// TwinCAT 3 PLC project STELLA1Runtime
// ProgramVersion: 3.1.4023.0
// libraries:
//   Tc2_DataExchange, * (Beckhoff Automation GmbH)
//   Tc2_Math, * (Beckhoff Automation GmbH)
//   Tc2_MC2, * (Beckhoff Automation GmbH)
//   Tc2_MC2_Drive, * (Beckhoff Automation GmbH)
//   Tc2_NC, * (Beckhoff Automation GmbH)
//   Tc2_Standard, * (Beckhoff Automation GmbH)
//   Tc2_System, * (Beckhoff Automation GmbH)
//   Tc2_Utilities, * (Beckhoff Automation GmbH)
//   Tc3_IotBase, * (Beckhoff Automation GmbH)
//   Tc3_Module, * (Beckhoff Automation GmbH)
//   VisuDialogs, * (System)
//   PS_DcUpsEC,2.0,Phoenix Contact GmbH & Co.KG
//   VisuSymbols,3.5.10.0,System
// project tree:
//   DUTs/ E_Blink.TcDUT (not stored), E_Horn.TcDUT (not stored), E_TCSCommand.TcDUT, E_TCSErrors.TcDUT, E_TelescopeMode.TcDUT (not stored)
//   / GlobalTextList.TcGTLO, PlcTask.TcTTO (not stored), Visualization Manager.TcVMO (not stored)
//   GVLs/ GVL_FilterWheel.TcGVL (not stored), GVL_Hydraulics.TcGVL, GVL_Main.TcGVL, GVL_pendant_control.TcGVL (not stored), GVL_Safety.TcGVL, GVL_Telescope.TcGVL (not stored)
//   POUs/ AzimuthElevationControl.TcPOU, CoverControl.TcPOU, DerotatorControl.TcPOU, ElevationControl.TcPOU, FilterWheelControl.TcPOU, FocusControl.TcPOU, HydraulicsControl.TcPOU, MAIN.TcPOU, NasmythControl.TcPOU (not stored), PendantControl.TcPOU (not stored), PowerMonitoring.TcPOU, SafetyHandling.TcPOU (not stored), TelescopeAuxiliary.TcPOU (not stored), TelescopeControl.TcPOU, Transformer.TcPOU
//   POUs/FunctionBlocks/ CO_ABERRATION.TcPOU, CO_NUTATE.TcPOU, CO_REFRACT.TcPOU (not stored), FB_ALTAZ2HADEC.TcPOU (not stored), FB_AstroClock.TcPOU, FB_Axis2.TcPOU, FB_BLINK.TcPOU, FB_ButtonEnable.TcPOU (not stored), FB_Cover.TcPOU (not stored), FB_CO_NUTATE.TcPOU (not stored), FB_EQ2HOR.TcPOU, FB_EQ2HOR2.TcPOU, FB_EventLog.TcPOU (not stored), FB_HADEC2ALTAZ.TcPOU (not stored), FB_HOR2EQ.TcPOU, FB_HOR2EQ2.TcPOU, FB_Horn.TcPOU, FB_InfluxMessage.TcPOU (not stored), FB_LightTimer.TcPOU, FB_MQTTCommunication.TcPOU, FB_NUTATE.TcPOU, FB_PRECESS.TcPOU (not stored), FB_PRECESS2.TcPOU (not stored), FB_PRECESS3.TcPOU, FB_RFTRIG.TcPOU (not stored), FB_SUNPOS.TcPOU, FB_TimeAverage.TcPOU, FB_Timer.TcPOU, FB_TONTP.TcPOU (not stored), TelescopeAxisClass.TcPOU (not stored)
//   POUs/Functions/ ATAN2.TcPOU, CO_REFRACT_FORWARD.TcPOU (not stored), CT2LST.TcPOU, DateTime2JD.TcPOU, F_Azimuthvelocity.TcPOU, F_DerotatorPosition2.TcPOU, F_Derotatorvelocity.TcPOU (not stored), F_Elevationvelocity.TcPOU, F_YREAL.TcPOU (not stored), NCError_TO_STRING.TcPOU, PointingModelAzimuth.TcPOU (not stored), PointingModelElevation.TcPOU (not stored), POLY.TcPOU, Refraction.TcPOU, TEN.TcPOU (not stored)
//   VISUs/ Visualization.TcVIS
// real-time tasks:
//   TASK PlcTask: cycle T#10ms, priority 20, ADS port 350
// motion (NC):
//   TASK NC-Task 1 SAF: cycle T#2ms, priority 4, ADS port 501
//   TASK NC-Task 1 SVB: cycle T#10ms, priority 8, ADS port 511
//   AXIS Fokus (id 1)
//     Dynamic: AccelerationMaximum=100, DecelerationMaximum=100, Acceleration=4.5, Deceleration=4.5, Jerk=13.5
//     Velo: RefSearch=0.2, RefSync=0.2, SlowManual=0.1, FastManual=0.5, Maximum=3
//     TargetPosControl: Range=0.1
//     OtherSettings: AllowMotionCmdToSlave=true, PulseDistancePos=1, PulseDistanceNeg=1
//     encoder EncType=4
//       EncPara: ScaleFactorNumerator=0.001, ScaleFactorDenominator=5, MaxCount=#x0000ffff
//         SoftEndMinControl: Enable=true
//         SoftEndMaxControl: Enable=true, Range=100
//         Inc: RefMode=2, RefSoftSyncMask=#x0000ffff
//     drive DrvType=23
//       Analog: VeloReferenz=10.2713178, VeloScale=10, TorqueSetpointScale=10, ScaleFactorActTorque=10
//       TimeComp: TaskDelayCycles=1
//     controller CtrType=1
//       CtrPara: PriorControlFactor=1
//         PosDiffControl: Range=1
//         PID: PosKp=12, CtrlOutputLimit=1
//         Observer: BandWidth=20
//   AXIS Derotator (id 2)
//     General: UnitName=°
//     Dynamic: AccelerationMaximum=20, DecelerationMaximum=20, Acceleration=3.70696, Deceleration=3.70696, Jerk=1.65107
//     Velo: RefSearch=1, RefSync=0.5, SlowManual=0.5, FastManual=5, Fast=11.7222517903646, Maximum=11.7223
//     PositionAreaControl: Range=10
//     TargetPosControl: Range=1, Time=0.1
//     OtherSettings: AllowMotionCmdToSlave=true
//     encoder EncType=8
//       EncPara: ScaleFactorNumerator=0.2, ScaleFactorDenominator=1048576, MaxCount=#xffffffff
//         SoftEndMinControl: Enable=true, Range=-70
//         SoftEndMaxControl: Enable=true, Range=380
//     drive DrvType=9
//       DrvPara: MaxCount=#xffffffff, DriveControlDWord=#x00030100
//         Analog: VeloReferenz=12.894476969401, TorqueSetpointScale=10, ScaleFactorActTorque=0.1
//         TimeComp: TaskDelayCycles=1
//     controller CtrType=1
//       CtrPara: PriorControlFactor=1
//         PosDiffControl: Range=1, Time=0.1
//         Observer: BandWidth=20
//   AXIS Azimuth (id 3)
//     General: UnitName=°
//     Dynamic: AccelerationMaximum=10, DecelerationMaximum=10, Acceleration=3, Deceleration=3, Jerk=1
//     Velo: RefSearch=2, RefSync=1, SlowManual=1, FastManual=5, Fast=798, Maximum=10
//     TargetPosControl: Range=1, Time=0.1
//     OtherSettings: AllowMotionCmdToSlave=true
//     encoder EncType=8
//       EncPara: ScaleFactorNumerator=360, ScaleFactorDenominator=1048576, MaxCount=#xffffffff
//         SoftEndMinControl: Enable=true, Range=-50
//         SoftEndMaxControl: Enable=true, Range=450
//         Inc: RefPosition=180, RefMode=2
//     drive DrvType=9
//       DrvPara: MaxCount=#xffffffff, DriveControlDWord=#x00030100
//         Analog: VeloReferenz=877.8, VeloScale=1.02400649589962, TorqueSetpointScale=10, ScaleFactorActTorque=0.1
//         TimeComp: TaskDelayCycles=1
//     controller CtrType=1
//       CtrPara: PriorControlFactor=1
//         PosDiffControl: Range=3, Time=0.1
//         Observer: BandWidth=20
//   AXIS Elevation (id 4)
//     General: UnitName=°
//     Dynamic: AccelerationMaximum=10, DecelerationMaximum=10, Acceleration=3, Deceleration=3, Jerk=2
//     Velo: RefSearch=0.5, RefSync=0.5, SlowManual=1, FastManual=3, Fast=1026, Maximum=10
//     TargetPosControl: Range=1, Time=0.1
//     OtherSettings: AllowMotionCmdToSlave=true
//     encoder EncType=8
//       EncPara: ScaleFactorNumerator=360, ScaleFactorDenominator=1048576, MaxCount=#xffffffff
//         SoftEndMinControl: Enable=true
//         SoftEndMaxControl: Enable=true, Range=91
//         Inc: RefPosition=73.9885, RefMode=2
//     drive DrvType=9
//       DrvPara: MaxCount=#xffffffff, DriveControlDWord=#x00030100
//         Analog: VeloReferenz=1128.6, VeloScale=1.02400649589962, TorqueSetpointScale=10, ScaleFactorActTorque=0.1
//         TimeComp: TaskDelayCycles=1
//     controller CtrType=1
//       CtrPara: PriorControlFactor=1
//         PosDiffControl: Range=1, Time=0.1
//         Observer: BandWidth=20
//   AXIS FilterWheel (id 5)
//     General: UnitName=°, UnitFlags=#x00000004
//     Dynamic: AccelerationMaximum=1500, DecelerationMaximum=1500, Acceleration=100, Deceleration=100, Jerk=100
//     Velo: RefSearch=5, RefSync=2.5, SlowManual=3, FastManual=30, Fast=207.666666666667, Maximum=207.667
//     TargetPosControl: Range=1
//     OtherSettings: AllowMotionCmdToSlave=true
//     encoder EncType=19
//       EncPara: ScaleFactorNumerator=10, ScaleFactorDenominator=1048576, MaxCount=#xffffffff
//         Inc: RefMode=1, HomingSensorSource=9
//     drive DrvType=16
//       DrvPara: MaxCount=#xffffffff, DriveControlDWord=#x00020000
//         Analog: VeloReferenz=228.433333333333, VeloScale=30, PosScale=10, TorqueSetpointScale=10, ScaleFactorActTorque=0.1
//         TimeComp: TaskDelayCycles=1
//     controller CtrType=1
//       CtrPara: PriorControlFactor=1
//         PosDiffControl: Enable=false, Range=0.2
//         PID: PosKp=5
//         Observer: BandWidth=20
// I/O:
//   DEVICE Gerät 1 (EtherCAT), AmsNetId 5.122.3.233.2.1
//     Klemme 30 (EK1200) [EK1200-5000 EtherCAT Netzteil (2A E-Bus)]
//       Safety Logic (EL6910) [EL6910, TwinSAFE PLC]
//       Safety IN (EL1904) [EL1904, 4 Ch. Safety Input 24V, TwinSAFE]
//         modules: Module 1 (FSOES)
//       Safety OUT (EL2904) [EL2904, 4 Ch. Safety Output 24V, 0.5A, TwinSAFE]
//         modules: Module 1 (FSOES), Module 2 (DO)
//       Power analysis (EL3443) [EL3443 3Ch. Power Measuring]
//       Power0 (EL9410) [EL9410 E-Bus Netzteilklemme (Diagnose)]
//       Main Panel IN (EL1008) [EL1008 8K. Dig. Eingang 24V, 3ms]
//       Hydraulics IN (EL1008) [EL1008 8K. Dig. Eingang 24V, 3ms]
//       Trafo Hydraulics IN (EL1008) [EL1008 8K. Dig. Eingang 24V, 3ms]
//       Main Panel Out (EL2008) [EL2008 8K. Dig. Ausgang 24V, 0.5A]
//       Trafo Hydraulics OUT (EL2008) [EL2008 8K. Dig. Ausgang 24V, 0.5A]
//       Temperature IN (EL3202) [EL3202 2K.Ana. Eingang PT100 (RTD)]
//       Power1 (EL9410) [EL9410 E-Bus Netzteilklemme (Diagnose)]
//       Pendant Control (EL1008) [EL1008 8K. Dig. Eingang 24V, 3ms]
//       Pendant Control2 (EL1008) [EL1008 8K. Dig. Eingang 24V, 3ms]
//       M2 M3 Limit switches (EL1008) [EL1008 8K. Dig. Eingang 24V, 3ms]
//       Cover Limit Switches (EL1008) [EL1008 8K. Dig. Eingang 24V, 3ms]
//       Telescope Hydraulics IN (EL1008) [EL1008 8K. Dig. Eingang 24V, 3ms]
//       Pendant Lights (EL2008) [EL2008 8K. Dig. Ausgang 24V, 0.5A]
//       Lock and Horn (EL2008) [EL2008 8K. Dig. Ausgang 24V, 0.5A]
//       Temperature M2 M1 (EL3064) [EL3064 4K.Ana. Eingang 0-10V]
//       Power2 (EL9410) [EL9410 E-Bus Netzteilklemme (Diagnose)]
//       FocusMotor (EL7342) [EL7342 2K. DC-Motor-Endstufe (50V, 3.5A)]
//       FocusEncoder (EL5101-0010) [EL5101-0010 1K. Inc. Encoder 5V (20 Mio. Inkremente/s)]
//       Cover Motors (EL2008) [EL2008 8K. Dig. Ausgang 24V, 0.5A]
//       Klemme 54 (EK1521) [EK1521 1-Port EtherCAT-Abzweig (FX-MultiMode)]
//         Klemme 55 (EK1501) [EK1501 EtherCAT-Koppler (2A E-Bus, FX-MultiMode, ID-Switch)]
//           FilterWheel (EL7211-0010) [EL7211-0010 1K. MDP742 Servo-Motor-Endstufe mit OCT (50V, 4,5A RMS)]
//           Klemme 57 (EL1008) [EL1008 8K. Dig. Eingang 24V, 3ms]
//           Klemme 58 (EL2008) [EL2008 8K. Dig. Ausgang 24V, 0.5A]
//           ShutterCOM (EL6001) [EL6001 Schnittstelle (RS232)]
//           Klemme 60 (EL3064) [EL3064 4K.Ana. Eingang 0-10V]
//           Klemme 69 (EL3202-0010) [EL3202-0010 2K. Ana. Eingang PT100 (RTD), hochgenau]
//           Klemme 65 (EL9011) [EL9011 Endklemme]
//       Klemme 61 (EK1110) [EK1110 EtherCAT-Verlängerung]
//     Derotator(AX5203-0000-0210) [AX5203-0000-0210 EtherCAT Drive (SoE, 2 Ch.)]
//     Azimuth (AX5125-0000-0214) [AX5125-0000-0214 EtherCAT Drive (SoE, 1 Ch.)]
//     Elevation (AX5125-0000-0214) [AX5125-0000-0214 EtherCAT Drive (SoE, 1 Ch.)]
//     Box 74 (Uninterruptible Power Supply) [QUINT4-UPS/24DC/24DC/40/EC]
// variable links:
//   Device 1 (EtherCAT) <-> Device 1 (EtherCAT)/Term 30 (EK1200)/Safety IN (EL1904)
//     Term 30 (EK1200)/Safety Logic (EL6910)/ConnectionOutputs/TwinSafeGroup1.Safety IN (EL1904) - Module 1 (FSOES)_10 RxPDO <-> Module 1 (FSOES)/TxPDO/FSOE
//   Device 1 (EtherCAT) <-> Device 1 (EtherCAT)/Term 30 (EK1200)/Safety Logic (EL6910)
//     Term 30 (EK1200)/Safety IN (EL1904)/Module 1 (FSOES)/RxPDO/FSOE <-> ConnectionInputs/TwinSafeGroup1.Safety IN (EL1904) - Module 1 (FSOES)_10 TxPDO
//     Term 30 (EK1200)/Safety OUT (EL2904)/Module 1 (FSOES)/TxPDO/FSOE <-> ConnectionOutputs/TwinSafeGroup1.Safety OUT (EL2904) - Module 1 (FSOES)_11 RxPDO
//   Device 1 (EtherCAT) <-> Device 1 (EtherCAT)/Term 30 (EK1200)/Safety OUT (EL2904)
//     Term 30 (EK1200)/Safety Logic (EL6910)/ConnectionInputs/TwinSafeGroup1.Safety OUT (EL2904) - Module 1 (FSOES)_11 TxPDO <-> Module 1 (FSOES)/RxPDO/FSOE
//   NC-Task 1 SAF/Axes/Azimuth <-> Device 1 (EtherCAT)/Azimuth (AX5125-0000-0214)
//     Drive/Inputs/In/nDataIn1 <-> AT/Following distance
//     Drive/Inputs/In/nDcOutputTime <-> InfoData/DcOutputShift
//     Drive/Inputs/In/nState1 <-> AT/Drive status word @bit 8
//     Drive/Inputs/In/nState2 <-> AT/Drive status word
//     Drive/Inputs/In/nState4 @bit 1 <-> WcState/InputToggle
//     Drive/Inputs/In/nState4 <-> WcState/WcState
//     Drive/Outputs/Out/nCtrl1 <-> MDT/Master control word @bit 8
//     Drive/Outputs/Out/nDataOut1 <-> MDT/Position command value
//     Enc/Inputs/In/nDataIn1 <-> AT/Position feedback 1 value
//     Enc/Inputs/In/nDataIn3 <-> AT/Probe value 1 positive edge
//     Enc/Inputs/In/nDcInputTime <-> InfoData/DcInputShift
//     Enc/Inputs/In/nState4 @bit 1 <-> WcState/InputToggle
//     Enc/Inputs/In/nState4 <-> WcState/WcState
//     Enc/Inputs/In/nState5 <-> AT/Probe 1 positive latched
//     Enc/Outputs/Out/nCtrl5 <-> MDT/Probe 1 enable
//   NC-Task 1 SAF/Axes/Derotator <-> Device 1 (EtherCAT)/Derotator(AX5203-0000-0210)
//     Drive/Inputs/In/nDataIn1 <-> AT 1/Following distance
//     Drive/Inputs/In/nDataIn3[0] <-> AT 1/Torque/force feedback value
//     Drive/Inputs/In/nDcOutputTime <-> InfoData/DcOutputShift
//     Drive/Inputs/In/nState1 <-> AT 1/Drive status word @bit 8
//     Drive/Inputs/In/nState2 <-> AT 1/Drive status word
//     Drive/Inputs/In/nState4 @bit 1 <-> WcState/InputToggle
//     Drive/Inputs/In/nState4 <-> WcState/WcState
//     Drive/Outputs/Out/nCtrl1 <-> MDT 1/Master control word @bit 8
//     Drive/Outputs/Out/nDataOut1 <-> MDT 1/Position command value
//     Enc/Inputs/In/nDataIn1 <-> AT 1/Position feedback 1 value
//     Enc/Inputs/In/nDcInputTime <-> InfoData/DcInputShift
//     Enc/Inputs/In/nState4 @bit 1 <-> WcState/InputToggle
//     Enc/Inputs/In/nState4 <-> WcState/WcState
//   NC-Task 1 SAF/Axes/Elevation <-> Device 1 (EtherCAT)/Elevation (AX5125-0000-0214)
//     Drive/Inputs/In/nDataIn1 <-> AT/Following distance
//     Drive/Inputs/In/nDcOutputTime <-> InfoData/DcOutputShift
//     Drive/Inputs/In/nState1 <-> AT/Drive status word @bit 8
//     Drive/Inputs/In/nState2 <-> AT/Drive status word
//     Drive/Inputs/In/nState4 @bit 1 <-> WcState/InputToggle
//     Drive/Inputs/In/nState4 <-> WcState/WcState
//     Drive/Outputs/Out/nCtrl1 <-> MDT/Master control word @bit 8
//     Drive/Outputs/Out/nDataOut1 <-> MDT/Position command value
//     Enc/Inputs/In/nDataIn1 <-> AT/Position feedback 1 value
//     Enc/Inputs/In/nDataIn3 <-> AT/Probe value 1 positive edge
//     Enc/Inputs/In/nDcInputTime <-> InfoData/DcInputShift
//     Enc/Inputs/In/nState4 @bit 1 <-> WcState/InputToggle
//     Enc/Inputs/In/nState4 <-> WcState/WcState
//     Enc/Inputs/In/nState5 <-> AT/Probe 1 positive latched
//     Enc/Outputs/Out/nCtrl5 <-> MDT/Probe 1 enable
//   NC-Task 1 SAF/Axes/FilterWheel <-> Device 1 (EtherCAT)/Term 30 (EK1200)/Term 54 (EK1521)/Term 55 (EK1501)/FilterWheel (EL7211-0010)
//     Drive/Inputs/In/nDcOutputTime <-> InfoData/DcOutputShift
//     Drive/Inputs/In/nState1 <-> DRV Statusword/Statusword
//     Drive/Inputs/In/nState2 <-> DRV Statusword/Statusword @bit 8
//     Drive/Inputs/In/nState4 @bit 1 <-> WcState/InputToggle
//     Drive/Inputs/In/nState4 <-> WcState/WcState
//     Drive/Inputs/In/nState8 <-> DRV Info data 1/Info data 1
//     Drive/Outputs/Out/nCtrl1 <-> DRV Controlword/Controlword
//     Drive/Outputs/Out/nCtrl2 <-> DRV Controlword/Controlword @bit 8
//     Drive/Outputs/Out/nDataOut2 <-> DRV Target velocity/Target velocity
//     Enc/Inputs/In/nDataIn1 <-> FB Position/Position
//     Enc/Inputs/In/nDcInputTime <-> InfoData/DcInputShift
//     Enc/Inputs/In/nState4 @bit 1 <-> WcState/InputToggle
//     Enc/Inputs/In/nState4 <-> WcState/WcState
//   NC-Task 1 SAF/Axes/Fokus <-> Device 1 (EtherCAT)/Term 30 (EK1200)/FocusEncoder (EL5101-0010)
//     Enc/Inputs/In/nDataIn1[0] <-> ENC Status compact/Counter value
//     Enc/Inputs/In/nDataIn2[0] <-> ENC Status compact/Latch value
//     Enc/Inputs/In/nState1 <-> ENC Status compact/Status/Latch C valid
//     Enc/Inputs/In/nState1 @bit 1 <-> ENC Status compact/Status/Latch extern valid
//     Enc/Inputs/In/nState1 @bit 6 <-> ENC Status compact/Status/Open circuit
//     Enc/Inputs/In/nState1 @bit 2 <-> ENC Status compact/Status/Set counter done
//     Enc/Inputs/In/nState1 @bit 5 <-> ENC Status compact/Status/Status of input status
//     Enc/Inputs/In/nState2 @bit 4 <-> ENC Status compact/Status/Status of extern latch
//     Enc/Inputs/In/nState2 <-> ENC Status compact/Status/Status of input A
//     Enc/Inputs/In/nState2 @bit 1 <-> ENC Status compact/Status/Status of input B
//     Enc/Inputs/In/nState2 @bit 2 <-> ENC Status compact/Status/Status of input C
//     Enc/Inputs/In/nState2 @bit 3 <-> ENC Status compact/Status/Status of input gate
//     Enc/Inputs/In/nState2 @bit 5 <-> ENC Status compact/Status/Sync error
//     Enc/Inputs/In/nState2 @bit 6 <-> ENC Status compact/Status/TxPDO State
//     Enc/Inputs/In/nState2 @bit 7 <-> ENC Status compact/Status/TxPDO Toggle
//     Enc/Inputs/In/nState4 @bit 1 <-> WcState/InputToggle
//     Enc/Inputs/In/nState4 <-> WcState/WcState
//     Enc/Outputs/Out/nCtrl1 <-> ENC Control compact/Control/Enable latch C
//     Enc/Outputs/Out/nCtrl1 @bit 3 <-> ENC Control compact/Control/Enable latch extern on negative edge
//     Enc/Outputs/Out/nCtrl1 @bit 1 <-> ENC Control compact/Control/Enable latch extern on positive edge
//     Enc/Outputs/Out/nCtrl1 @bit 2 <-> ENC Control compact/Control/Set counter
//     Enc/Outputs/Out/nDataOut1[0] <-> ENC Control compact/Set counter value
//   NC-Task 1 SAF/Axes/Fokus <-> Device 1 (EtherCAT)/Term 30 (EK1200)/FocusMotor (EL7342)
//     Drive/Inputs/In/nState1 @bit 3 <-> DCM Status Channel 1/Status/Error
//     Drive/Inputs/In/nState1 @bit 5 <-> DCM Status Channel 1/Status/Moving negative
//     Drive/Inputs/In/nState1 @bit 4 <-> DCM Status Channel 1/Status/Moving positive
//     Drive/Inputs/In/nState1 @bit 1 <-> DCM Status Channel 1/Status/Ready
//     Drive/Inputs/In/nState1 <-> DCM Status Channel 1/Status/Ready to enable
//     Drive/Inputs/In/nState1 @bit 6 <-> DCM Status Channel 1/Status/Torque reduced
//     Drive/Inputs/In/nState1 @bit 2 <-> DCM Status Channel 1/Status/Warning
//     Drive/Inputs/In/nState2 @bit 3 <-> DCM Status Channel 1/Status/Digital input 1
//     Drive/Inputs/In/nState2 @bit 4 <-> DCM Status Channel 1/Status/Digital input 2
//     Drive/Inputs/In/nState2 @bit 5 <-> DCM Status Channel 1/Status/Sync error
//     Drive/Inputs/In/nState2 @bit 7 <-> DCM Status Channel 1/Status/TxPDO Toggle
//     Drive/Inputs/In/nState4 @bit 1 <-> WcState/InputToggle
//     Drive/Inputs/In/nState4 <-> WcState/WcState
//     Drive/Outputs/Out/nCtrl1 <-> DCM Control Channel 1/Control/Enable
//     Drive/Outputs/Out/nCtrl1 @bit 2 <-> DCM Control Channel 1/Control/Reduce torque
//     Drive/Outputs/Out/nCtrl1 @bit 1 <-> DCM Control Channel 1/Control/Reset
//     Drive/Outputs/Out/nCtrl1 @bit 3 <-> DCM Control Channel 1/Control/Threshold active
//     Drive/Outputs/Out/nDataOut2[0] <-> DCM Velocity Channel 1/Velocity
//   STELLA1Runtime/STELLA1Runtime Instance <-> Device 1 (EtherCAT)/Azimuth (AX5125-0000-0214)
//     PlcTask Inputs/GVL_Telescope.Azimuth_diagnostic <-> AT/Diagnostic number
//     PlcTask Inputs/GVL_Telescope.Azimuth_inputs <-> AT/Digital inputs, state
//     PlcTask Inputs/GVL_Telescope.Azimuth_torque <-> AT/Torque/force feedback value
//   STELLA1Runtime/STELLA1Runtime Instance <-> Device 1 (EtherCAT)/Box 74 (Uninterruptible Power Supply)
//     PlcTask Inputs/MAIN.arrInputPD @bit {304..432 step 32} <-> TxPDO 1/BATTERY {1..5} ALARMS  (5 links)
//     PlcTask Inputs/MAIN.arrInputPD @bit 80 <-> TxPDO 1/STATUS ACTUAL INPUT CURRENT
//     PlcTask Inputs/MAIN.arrInputPD @bit 64 <-> TxPDO 1/STATUS ACTUAL INPUT VOLTAGE
//     PlcTask Inputs/MAIN.arrInputPD @bit 112 <-> TxPDO 1/STATUS ACTUAL OUTPUT CURRENT 1
//     PlcTask Inputs/MAIN.arrInputPD @bit 96 <-> TxPDO 1/STATUS ACTUAL OUTPUT VOLTAGE 1
//     PlcTask Inputs/MAIN.arrInputPD @bit 128 <-> TxPDO 1/STATUS BATTERY ACTUAL VOLTAGE
//     PlcTask Inputs/MAIN.arrInputPD @bit 144 <-> TxPDO 1/STATUS BATTERY CHARGE CURRENT
//     PlcTask Inputs/MAIN.arrInputPD @bit 160 <-> TxPDO 1/STATUS BATTERY TEMPERATURE
//     PlcTask Inputs/MAIN.arrInputPD @bit 176 <-> TxPDO 1/STATUS DEVICE TEMPERATURE
//     PlcTask Inputs/MAIN.arrInputPD <-> TxPDO 1/STATUS FUNCTIONS
//     PlcTask Inputs/MAIN.arrInputPD @bit 32 <-> TxPDO 1/STATUS INTERFACE
//     PlcTask Inputs/MAIN.arrInputPD @bit 192 <-> TxPDO 1/STATUS SOC REMAINING TIME
//     PlcTask Inputs/MAIN.arrInputPD @bit 224 <-> TxPDO 1/STATUS SOC REMAINING TIME PC SHUTDOWN
//     PlcTask Inputs/MAIN.arrInputPD @bit 240 <-> TxPDO 1/STATUS SOH REMAINING LIFETIME
//     PlcTask Inputs/MAIN.arrInputPD @bit 272 <-> TxPDO 1/UPS DIAGNOSIS ALARMS
//     PlcTask Inputs/MAIN.arrInputPD @bit 256 <-> TxPDO 1/UPS PROCESS ALARMS
//   STELLA1Runtime/STELLA1Runtime Instance <-> Device 1 (EtherCAT)/Derotator(AX5203-0000-0210)
//     PlcTask Inputs/GVL_Telescope.Derotator_diagnostic <-> AT 1/Diagnostic number
//     PlcTask Inputs/GVL_Telescope.Derotator_inputs <-> AT 1/Digital inputs, state
//     PlcTask Inputs/GVL_Telescope.Derotator_torque <-> AT 1/Torque/force feedback value
//   STELLA1Runtime/STELLA1Runtime Instance <-> Device 1 (EtherCAT)/Elevation (AX5125-0000-0214)
//     PlcTask Inputs/GVL_Telescope.Elevation_diagnostic <-> AT/Diagnostic number
//     PlcTask Inputs/GVL_Telescope.Elevation_inputs <-> AT/Digital inputs, state
//     PlcTask Inputs/GVL_Telescope.Elevation_torque <-> AT/Torque/force feedback value
//   STELLA1Runtime/STELLA1Runtime Instance <-> Device 1 (EtherCAT)/Term 30 (EK1200)/Cover Limit Switches (EL1008)
//     PlcTask Inputs/GVL_Telescope.cover1_closed <-> Channel 2/GVL_Telescope.cover1_closed
//     PlcTask Inputs/GVL_Telescope.cover2_closed <-> Channel 4/GVL_Telescope.cover2_closed
//     PlcTask Inputs/GVL_Telescope.cover3_closed <-> Channel 6/GVL_Telescope.cover3_closed
//     PlcTask Inputs/GVL_Telescope.cover1_open <-> Channel 1/GVL_Telescope.cover1_open
//     PlcTask Inputs/GVL_Telescope.cover2_open <-> Channel 3/GVL_Telescope.cover2_open
//     PlcTask Inputs/GVL_Telescope.cover3_open <-> Channel 5/GVL_Telescope.cover3_open
//   STELLA1Runtime/STELLA1Runtime Instance <-> Device 1 (EtherCAT)/Term 30 (EK1200)/Cover Motors (EL2008)
//     PlcTask Outputs/GVL_Telescope.close_cover1 <-> Channel 4/GVL_Telescope.close_cover1
//     PlcTask Outputs/GVL_Telescope.close_cover2 <-> Channel 6/GVL_Telescope.close_cover2
//     PlcTask Outputs/GVL_Telescope.close_cover3 <-> Channel 8/GVL_Telescope.close_cover3
//     PlcTask Outputs/GVL_Telescope.nasmyth_left <-> Channel 1/GVL_Telescope.nasmyth_left
//     PlcTask Outputs/GVL_Telescope.nasmyth_right <-> Channel 2/GVL_Telescope.nasmyth_right
//     PlcTask Outputs/GVL_Telescope.open_cover1 <-> Channel 3/GVL_Telescope.open_cover1
//     PlcTask Outputs/GVL_Telescope.open_cover2 <-> Channel 5/GVL_Telescope.open_cover2
//     PlcTask Outputs/GVL_Telescope.open_cover3 <-> Channel 7/GVL_Telescope.open_cover3
//   STELLA1Runtime/STELLA1Runtime Instance <-> Device 1 (EtherCAT)/Term 30 (EK1200)/Hydraulics IN (EL1008)
//     PlcTask Inputs/GVL_Hydraulics.oil_high <-> Channel 2/GVL_Hydraulics.oil_high
//     PlcTask Inputs/GVL_Hydraulics.oil_low <-> Channel 1/GVL_Hydraulics.oil_low
//     PlcTask Inputs/GVL_Hydraulics.oil_overtemperature <-> Channel 4/GVL_Hydraulics.oil_overtemperature
//     PlcTask Inputs/GVL_Hydraulics.oil_pressure_OK <-> Channel 3/GVL_Hydraulics.oil_pressure_OK
//     PlcTask Inputs/GVL_Hydraulics.oil_undertemperature <-> Channel 5/GVL_Hydraulics.oil_undertemperature
//     PlcTask Inputs/GVL_Hydraulics.oilfilter_dirty <-> Channel 6/GVL_Hydraulics.oilfilter_dirty
//   STELLA1Runtime/STELLA1Runtime Instance <-> Device 1 (EtherCAT)/Term 30 (EK1200)/Lock and Horn (EL2008)
//     PlcTask Outputs/GVL_Telescope.focus_unlock <-> Channel 1/GVL_Telescope.focus_lock
//     PlcTask Outputs/GVL_Telescope.horn <-> Channel 8/GVL_Telescope.horn
//     PlcTask Outputs/GVL_Telescope.nasmyth_lock <-> Channel 2/GVL_Telescope.nasmyth_lock
//   STELLA1Runtime/STELLA1Runtime Instance <-> Device 1 (EtherCAT)/Term 30 (EK1200)/M2 M3 Limit switches (EL1008)
//     PlcTask Inputs/GVL_Telescope.focus_limit_far <-> Channel 2/GVL_Telescope.focus_limit_far
//     PlcTask Inputs/GVL_Telescope.focus_limit_near <-> Channel 1/GVL_Telescope.focus_limit_near
//     PlcTask Inputs/GVL_Telescope.nasmyth_limit_left <-> Channel 3/GVL_Telescope.nasmyth_limit_left
//     PlcTask Inputs/GVL_Telescope.nasmyth_limit_right <-> Channel 4/GVL_Telescope.nasmyth_limit_right
//   STELLA1Runtime/STELLA1Runtime Instance <-> Device 1 (EtherCAT)/Term 30 (EK1200)/Main Panel IN (EL1008)
//     PlcTask Inputs/GVL_Main.key_switch_remote <-> Channel 1/GVL_Main.key_switch_remote
//     PlcTask Inputs/GVL_Main.reset_switch <-> Channel 4/GVL_Main.reset_switch
//     PlcTask Inputs/GVL_Main.start_switch <-> Channel 2/GVL_Main.start_switch
//     PlcTask Inputs/GVL_Main.stop_switch <-> Channel 3/GVL_Main.stop_switch
//   STELLA1Runtime/STELLA1Runtime Instance <-> Device 1 (EtherCAT)/Term 30 (EK1200)/Main Panel Out (EL2008)
//     PlcTask Outputs/GVL_Main.lamp_error <-> Channel 3/GVL_Main.lamp_error
//     PlcTask Outputs/GVL_Main.lamp_on_manual <-> Channel 2/GVL_Main.lamp_ready
//     PlcTask Outputs/GVL_Main.lamp_power <-> Channel 1/GVL_Main.lamp_power
//   STELLA1Runtime/STELLA1Runtime Instance <-> Device 1 (EtherCAT)/Term 30 (EK1200)/Pendant Control (EL1008)
//     PlcTask Inputs/GVL_pendant_control.BCD1 <-> Channel 1/GVL_pendant_control.BCD1
//     PlcTask Inputs/GVL_pendant_control.BCD2 <-> Channel 2/GVL_pendant_control.BCD2
//     PlcTask Inputs/GVL_pendant_control.BCD4 <-> Channel 3/GVL_pendant_control.BCD4
//     PlcTask Inputs/GVL_pendant_control.BCD8 <-> Channel 4/GVL_pendant_control.BCD8
//     PlcTask Inputs/GVL_pendant_control.direction_down <-> Channel 7/GVL_pendant_control.direction_down
//     PlcTask Inputs/GVL_pendant_control.direction_up <-> Channel 6/GVL_pendant_control.direction_up
//     PlcTask Inputs/GVL_pendant_control.key_switch <-> Channel 8/GVL_pendant_control.key_switch
//     PlcTask Inputs/GVL_pendant_control.reset_switch <-> Channel 5/GVL_pendant_control.reset_switch
//   STELLA1Runtime/STELLA1Runtime Instance <-> Device 1 (EtherCAT)/Term 30 (EK1200)/Pendant Control2 (EL1008)
//     PlcTask Inputs/GVL_pendant_control.direction_left <-> Channel 2/GVL_pendant_control.direction_left
//     PlcTask Inputs/GVL_pendant_control.direction_right <-> Channel 3/GVL_pendant_control.direction_right
//     PlcTask Inputs/GVL_pendant_control.start_switch <-> Channel 1/GVL_pendant_control.start_switch
//   STELLA1Runtime/STELLA1Runtime Instance <-> Device 1 (EtherCAT)/Term 30 (EK1200)/Pendant Lights (EL2008)
//     PlcTask Outputs/GVL_pendant_control.lamp_down <-> Channel 2/GVL_pendant_control.lamp_down
//     PlcTask Outputs/GVL_pendant_control.lamp_error <-> Channel 5/GVL_pendant_control.lamp_error
//     PlcTask Outputs/GVL_pendant_control.lamp_left <-> Channel 4/GVL_pendant_control.lamp_left
//     PlcTask Outputs/GVL_pendant_control.lamp_right <-> Channel 3/GVL_pendant_control.lamp_right
//     PlcTask Outputs/GVL_pendant_control.lamp_up <-> Channel 1/GVL_pendant_control.lamp_up
//   STELLA1Runtime/STELLA1Runtime Instance <-> Device 1 (EtherCAT)/Term 30 (EK1200)/Power analysis (EL3443)
//     PlcTask Inputs/GVL_Main.ActiveEnergy <-> Total Active/Active Energy
//     PlcTask Inputs/GVL_Main.ActivePower <-> Total Active/Active Power
//     PlcTask Inputs/GVL_Main.NeutralLineCurrent <-> Total Basic/Calculated Neutral Line Current
//   STELLA1Runtime/STELLA1Runtime Instance <-> Device 1 (EtherCAT)/Term 30 (EK1200)/Safety Logic (EL6910)
//     PlcTask Inputs/GVL_Safety.Error <-> StandardInputs/TwinSafeGroup1.SafetyError_4
//     PlcTask Inputs/GVL_Safety.State <-> Function Block Info Data/TwinSafeGroup1.Network1.FBEstop1 Info Data/State
//     PlcTask Inputs/GVL_Safety.Stop <-> StandardInputs/TwinSafeGroup1.SafetyStop_7
//     PlcTask Outputs/GVL_Safety.ErrAck <-> StandardOutputs/TwinSafeGroup1.ErrorAcknowledgement_1
//     PlcTask Outputs/GVL_Safety.Restart <-> StandardOutputs/TwinSafeGroup1.RestartSafety_2
//     PlcTask Outputs/GVL_Safety.Run <-> StandardOutputs/TwinSafeGroup1.RunSafety_3
//   STELLA1Runtime/STELLA1Runtime Instance <-> Device 1 (EtherCAT)/Term 30 (EK1200)/Telescope Hydraulics IN (EL1008)
//     PlcTask Inputs/GVL_Hydraulics.oil_reserve <-> Channel 2/GVL_Hydraulics.oil_reserve
//     PlcTask Inputs/GVL_Hydraulics.oilpan_maximum <-> Channel 1/GVL_Hydraulics.oilpan_maximum
//     PlcTask Inputs/GVL_Telescope.azimut_limit_switch <-> Channel 8/GVL_Telescope.azimut_limit_switch
//   STELLA1Runtime/STELLA1Runtime Instance <-> Device 1 (EtherCAT)/Term 30 (EK1200)/Temperature IN (EL3202)
//     PlcTask Inputs/GVL_Main.main_cabinet_temperature <-> RTD Inputs Channel 1/Value
//   STELLA1Runtime/STELLA1Runtime Instance <-> Device 1 (EtherCAT)/Term 30 (EK1200)/Temperature M2 M1 (EL3064)
//     PlcTask Inputs/GVL_Hydraulics.oil_level <-> AI Standard Channel 3/GVL_Hydraulics.oil_level
//     PlcTask Inputs/GVL_Telescope.temperature_mirror1 <-> AI Standard Channel 2/GVL_Telescope.temperature_mirror1
//     PlcTask Inputs/GVL_Telescope.temperature_mirror2 <-> AI Standard Channel 1/GVL_Telescope.temperature_mirror2
//   STELLA1Runtime/STELLA1Runtime Instance <-> Device 1 (EtherCAT)/Term 30 (EK1200)/Term 54 (EK1521)/Term 55 (EK1501)/FilterWheel (EL7211-0010)
//     PlcTask Inputs/GVL_FilterWheel.bCalibrationCam <-> DRV Info data 1/Info data 1
//   STELLA1Runtime/STELLA1Runtime Instance <-> Device 1 (EtherCAT)/Term 30 (EK1200)/Term 54 (EK1521)/Term 55 (EK1501)/Term 60 (EL3064)
//     PlcTask Inputs/TelescopeAuxiliary.raw_dewar_pressure <-> AI Standard Channel 1/Value
//   STELLA1Runtime/STELLA1Runtime Instance <-> Device 1 (EtherCAT)/Term 30 (EK1200)/Trafo Hydraulics IN (EL1008)
//     PlcTask Inputs/GVL_Hydraulics.pump_running <-> Channel 7/GVL_Hydraulics.pump_running
//     PlcTask Inputs/GVL_Hydraulics.suction_running <-> Channel 8/GVL_Hydraulics.suction_running
//     PlcTask Inputs/GVL_Main.brake_clearing <-> Channel 3/GVL_Main.brake_clearing
//     PlcTask Inputs/GVL_Main.trafo_bypassed <-> Channel 2/GVL_Main.trafo_bypassed
//   STELLA1Runtime/STELLA1Runtime Instance <-> Device 1 (EtherCAT)/Term 30 (EK1200)/Trafo Hydraulics OUT (EL2008)
//     PlcTask Outputs/GVL_Hydraulics.oil_pump_enable <-> Channel 1/GVL_Hydraulics.oil_pump_enable
//     PlcTask Outputs/GVL_Hydraulics.oil_suction_enable <-> Channel 2/GVL_Hydraulics.oil_suction_enable
//     PlcTask Outputs/GVL_Main.softstart_trafo <-> Channel 8/GVL_Main.softstart_trafo
//     PlcTask Outputs/GVL_Telescope.brake_azimuth_eve <-> Channel 3/GVL_Telescope.brake_azimuth_eve
//   STELLA1Runtime/STELLA1Runtime Instance <-> NC-Task 1 SAF/Axes/Azimuth
//     PlcTask Inputs/GVL_Telescope.AzimuthAxisRef.NcToPlc <-> Outputs/ToPlc
//     PlcTask Outputs/GVL_Telescope.AzimuthAxisRef.PlcToNc <-> Inputs/FromPlc
//   STELLA1Runtime/STELLA1Runtime Instance <-> NC-Task 1 SAF/Axes/Derotator
//     PlcTask Inputs/GVL_Telescope.DerotatorAxisRef.NcToPlc <-> Outputs/ToPlc
//     PlcTask Outputs/GVL_Telescope.DerotatorAxisRef.PlcToNc <-> Inputs/FromPlc
//   STELLA1Runtime/STELLA1Runtime Instance <-> NC-Task 1 SAF/Axes/Elevation
//     PlcTask Inputs/GVL_Telescope.ElevationAxisRef.NcToPlc <-> Outputs/ToPlc
//     PlcTask Outputs/GVL_Telescope.ElevationAxisRef.PlcToNc <-> Inputs/FromPlc
//   STELLA1Runtime/STELLA1Runtime Instance <-> NC-Task 1 SAF/Axes/FilterWheel
//     PlcTask Inputs/GVL_FilterWheel.FilterWheel_AxisRef.NcToPlc <-> Outputs/ToPlc
//     PlcTask Outputs/GVL_FilterWheel.FilterWheel_AxisRef.PlcToNc <-> Inputs/FromPlc
//   STELLA1Runtime/STELLA1Runtime Instance <-> NC-Task 1 SAF/Axes/Fokus
//     PlcTask Inputs/GVL_Telescope.FocusAxisRef.NcToPlc <-> Outputs/ToPlc
//     PlcTask Outputs/GVL_Telescope.FocusAxisRef.PlcToNc <-> Inputs/FromPlc

// ---- DUTs/E_TCSCommand.TcDUT
{attribute 'qualified_only'}
{attribute 'strict'}
TYPE E_TCSCommand :
(
	no_command := 0,
	gohome,
	park,
	track,
	goto,
	stop,
	slew,
	poweron
);
END_TYPE

// ---- DUTs/E_TCSErrors.TcDUT
{attribute 'qualified_only'}
{attribute 'strict'}
TYPE E_TCSErrors :
(
	no_error := 0,
	info :=1,
	warning := 2,
    error := 4,
	panic := 8
);
END_TYPE

// ---- GVLs/GVL_Hydraulics.TcGVL
{attribute 'qualified_only'}
VAR_GLOBAL
	// 2.1
	oil_low				AT%I*: BOOL;
	// ?
	oil_high			AT%I*: BOOL;
	// 2.3
	oil_pressure_OK		AT%I*: BOOL;
	// 2.4
	oil_overtemperature		AT%I*: BOOL;
	// 2.5
	oil_undertemperature	AT%I*: BOOL;
	// 2.6
	oilfilter_dirty		AT%I*: BOOL;
	// 2.7
	pump_running		AT%I*: BOOL;
	// 2.8
	suction_running		AT%I*: BOOL;
	//BT2
	oil_level			AT%I*: INT;
	
	//DIN39 4.6
	oilpan_maximum		AT%I*: BOOL;
	//DIN40 4.7
	oil_reserve			AT%I*: BOOL;
	
		
	//DOUT4 0.3
	oil_pump_enable		AT%Q*: BOOL;
	//DOUT5 0.4
	oil_suction_enable		AT%Q*: BOOL;	
END_VAR

// ---- GVLs/GVL_Main.TcGVL
{attribute 'qualified_only'}
//TODO update to current RoboTel IOs
VAR_GLOBAL
	//DIN1 0.0
	//phase_available		AT%I*: BOOL;
	// not implemented on stella
	trafo_bypassed		AT%I*: BOOL;
	//not implemented on RoboTel
	//key_switch			AT%I*: BOOL;
	//DIN3 0.2
	key_switch_remote	AT%I*: BOOL;
	//DIN4 0.3
	start_switch		AT%I*: BOOL;
	//DIN5 0.4
	stop_switch			AT%I*: BOOL;
	//DIN8 0.7
	reset_switch		AT%I*: BOOL;
	
	//BT1
	main_cabinet_temperature	AT%I*: INT;
	//DIN15 1.6
	brake_clearing		AT%I*: BOOL;
	
	//DOUT1 0.0
	lamp_power			AT%Q*: BOOL;
	//DOUT2 0.1
	lamp_on_manual			AT%Q*: BOOL;
	//DOUT3 0.2
	lamp_error			AT%Q*: BOOL;
	
	//DOUT7 0.6
	softstart_trafo		AT%Q*:BOOL;

	isRoboTel:		BOOL;
	(*
	NeutralCurrentGuardWarning		AT%I*:	BOOL;
	NeutralCurrentGuarError			AT%I*:	BOOL;
	ActivePowerGuardWarning			AT%I*:	BOOL;
	ActivePowerGuardError			AT%I*:	BOOL;
	ApparentPowerGuardWarning		AT%I*:	BOOL;
	ApparentPowerGuardError			AT%I*:	BOOL;
	*)
END_VAR

// ---- GVLs/GVL_Safety.TcGVL
{attribute 'qualified_only'}
VAR_GLOBAL
	// Safety Error Condition
	Error		AT%I*:	BOOL;
	// Run/Stop Safety
	Run			AT%Q*:	BOOL;
	// Restart Safety
	Restart		AT%Q*:	BOOL;
	// Error Acknowledgement 
	ErrAck		AT%Q*:	BOOL;
	// Stop signal coming from Safety
	Stop		AT%I*:	BOOL;
	// state variable
	State		AT%I*:	USINT;
END_VAR

// ---- POUs/AzimuthElevationControl.TcPOU
PROGRAM AzimuthElevationControl
VAR_INPUT
	// enable the axis and its position control loop
	Enable:		BOOL;
	// reset the axis
	Reset: 		BOOL;
	// decrease azimuth
	left:		BOOL;
	// increase azimuth
	right: 		BOOL;
	// Move azimuth to given position
	MoveAxis:	BOOL;
	// Home the axis
	HomeAxis:	BOOL;
	// enable tracking
	Tracking:	BOOL;
	// position to move the axis to
	position: 	LREAL;
	// set the Velocity of the axis
	velocity:	LREAL;
	// stop the Axis
	StopAxis:	BOOL;
	// diagnostic reset
	bSoEReset:	BOOL;
END_VAR
VAR_OUTPUT
	// error state of the axis
	error: 			BOOL;
	// error ID of the axis
	ErrorID:		UDINT;
	// actual_position of the axis
	act_position:	LREAL;
	// is the axis calibrated
	calibrated:		BOOL;
	// drive is ready
	ready:			BOOL;
	// time to reach target position
	slewtime:		LREAL;
END_VAR
VAR
	AzimuthAxis:		FB_Axis2;
	AzimuthCalibration: MC_SetPosition;
	//fbSoEReset:			FB_SoEReset;
	AzimuthAxisEvent: 	FB_EventLog;
	AzimuthDiagnosticEvent: 	FB_EventLog;
	// delay until commutator angle is measured
	readydelay:			TON;
	HomeDelay:			FB_TONTP;
	TorqueError:		TON := (PT := T#3S);
	azimuth_torque: 	REAL;
	TorqueWarning:		FB_EventLog;
	CalibrationEvent:	FB_Eventlog;
	ReadParameter:		MC_ReadParameter;
	getlastposition:	BOOL := TRUE;
	azimuth_rest_timer:	TON;
	azimuth_at_rest:	BOOL;
	fbSoEReset: 		FB_SoEReset;
	DiagnosticError:	BOOL;
END_VAR
VAR CONSTANT
	// reference position for homing
	// homing_position:		LREAL := 439.0; // was 442 - -21.21 = 463.21; 463 + 24 = 439
	// current position of the calibration cam encoder zero index. Apply an offset here if necessary
	calibration_position:	LREAL :=  208.5009; //208.4983 - -0.0026;//208.6273; //208.6073; // 208.7122869;//207.0092; // 208.2342; 
END_VAR
VAR PERSISTENT
	last_position:	LREAL := -51.0;
END_VAR

(* Azimuth Axis control section
Power must be on and brake must be open for the axis to operate
*)

// generate the ready signal after enabling the drive
readydelay(IN :=  AzimuthAxis.Enable, PT := T#3000MS, Q=> ready);

// limit the input position angle
position := LIMIT(-50.0, position, 450.0);

// conduct the calibrated signal
calibrated := AzimuthAxis.Calibrated;

IF Calibrated OR Error THEN
	HomeAxis := FALSE;
	getlastposition := FALSE;
END_IF
	
IF HomeAxis THEN
	position := calibration_position;
END_IF

IF HomeDelay.Q THEN
	position := calibration_position;
	MoveAxis := TRUE;
END_IF

// perform a recalibration on the last known position
AzimuthCalibration(
	Axis := GVL_Telescope.AzimuthAxisRef,
	Execute := getlastposition AND last_position>=-50.0 AND NOT Calibrated,
	Position := last_position);

IF AzimuthCalibration.Done THEN
	getlastposition := FALSE;
END_IF

IF Calibrated THEN
	last_position := act_position;
END_IF

// enable the azimuth if not moved by the power chain. Sorry for the hack
azimuth_rest_timer(IN := HydraulicsControl.brake_open AND 
				(ABS(GVL_Telescope.AzimuthAxisRef.NcToPlc.ActVelo) < 0.01), PT := T#2S);
// if azimuth at rest or calibrated, allow enabling the azimuth
IF azimuth_rest_timer.Q or calibrated THEN
	azimuth_at_rest := TRUE;
ELSIF HydraulicsControl.brake_closed THEN
	azimuth_at_rest := FALSE;
END_IF
	
// deactivate limit switches on homing
MC_SetAcceptBlockedDriveSignal(
	Axis := GVL_Telescope.AzimuthAxisRef, 
	Enable := HomeAxis);

AzimuthAxis(	
	Enable := 			enable AND azimuth_at_rest AND NOT GVL_Telescope.azimut_limit_switch,
	Reset := 			reset,
	MoveAxis :=			MoveAxis,
	HomeAxis := 		HomeAxis,
	StopAxis :=			StopAxis,
	Tracking :=			Tracking,
	Position := 		position, 
	Velocity :=			velocity,
	Enable_Positive := 	GVL_Telescope.Azimuth_inputs.1 OR HomeAxis,
	Enable_Negative := 	GVL_Telescope.Azimuth_inputs.0,
	Jog_Forward :=		right,
	Jog_Backwards := 	left,
	bCalibrationCam :=	NOT GVL_Telescope.Azimuth_inputs.1,
	ActualPosition => 	act_position,
	Error => 			error,
	ErrorID => 			ErrorID,
	AxisRef :=			GVL_Telescope.AzimuthAxisRef);

IF bSoEReset THEN
	last_position := -51.0;
	fbSoEReset(
		Axis := GVL_Telescope.AzimuthAxisRef,
		Execute := TRUE,
		Timeout := DEFAULT_ADS_TIMEOUT);
 	IF fbSoEReset.Busy THEN
		fbSoEReset(Axis := GVL_Telescope.AzimuthAxisRef, Execute := FALSE);
	ELSE
		bSoEReset := FALSE;
		Reset := TRUE;
	END_IF
END_IF 

IF AzimuthAxis.MoveDone THEN
	MoveAxis := FALSE;
END_IF

IF AzimuthAxis.HomeDone THEN
	HomeAxis := FALSE;
END_IF
	
IF AzimuthAxis.ResetDone THEN
	reset := FALSE;
END_IF

IF AzimuthAxis.StopDone THEN
	StopAxis := FALSE;
END_IF
DiagnosticError := FALSE;
IF GVL_Telescope.Azimuth_diagnostic < 16#D012 AND GVL_Telescope.Azimuth_diagnostic > 16#D014 THEN
	DiagnosticError :=TRUE;
	ErrorID := GVL_Telescope.Azimuth_diagnostic;
END_IF

ReadParameter(	Axis := GVL_Telescope.AzimuthAxisRef, Enable := AzimuthAxis.InMotion, 
				ParameterNumber := MC_AxisParameter.AxisRemainingTimeToGo, 
				ReadMode := E_ReadMode.READMODE_CYCLIC);
IF ReadParameter.Valid THEN
	slewtime := ReadParameter.Value;
END_IF

azimuth_torque := GVL_Telescope.Azimuth_torque / 10.0;
TorqueError(IN := ABS(azimuth_torque) > 50.0);


AzimuthAxisEvent(	
	Trigger := 		Error, 
	Level := 		ADSLOG_MSGTYPE_ERROR,
	FormatString :=	'Azimuth Axis Error: %s',
	OnMessage := 	NCError_TO_STRING(ErrorID));
	
AzimuthDiagnosticEvent(	
	Trigger := 		DiagnosticError,
	Level := 		ADSLOG_MSGTYPE_ERROR,
	FormatString :=	'Azimuth Axis Diagnostic Error: %s',
	OnMessage := 	NCError_TO_STRING(GVL_Telescope.Azimuth_diagnostic));
	
TorqueWarning(	
	Trigger := 		TorqueError.Q, 
	Level := 		ADSLOG_MSGTYPE_WARN,
	FormatString :=	'%s',
	OnMessage := 	'Azimuth torque is high.');
	
CalibrationEvent(
	Trigger := 		Calibrated, 
	Level := 		ADSLOG_MSGTYPE_HINT,
	FormatString :=	'%s',
	OnMessage := 	'Azimuth axis is calibrated.');

END_PROGRAM

// ---- POUs/FunctionBlocks/FB_Axis2.TcPOU
FUNCTION_BLOCK FB_Axis2
VAR_INPUT
	// enable the axis
	Enable:		BOOL;
	// reset the axis after error
	Reset: 		BOOL;
	// Move the Axis to a given position
	MoveAxis: 	BOOL;
	// HomeAxis;
	HomeAxis:	BOOL;
	// Stop the axis
	StopAxis:	BOOL;
	// position to move to
	Position: 	LREAL;
	// maximum velocity
	Velocity:	LREAL := 10.0;
	// Enable movement in positive direction (considering limit switch)
	Enable_Positive:	BOOL := TRUE;
	// Enable movement in negative direction (considering limit switch)
	Enable_Negative:	BOOL := TRUE;
	// jog forward
	Jog_Forward:		BOOL := FALSE;
	// jog backward
	Jog_Backwards:		BOOL := FALSE;
	// calibration input for homing
	bCalibrationCam:	BOOL;
	isModuloAxis:		BOOL := FALSE;
	// enable external setpoint generator
	Tracking:			BOOL;
	HomingMode:			MC_HomingMode := MC_HomingMode.MC_DefaultHoming;
END_VAR
VAR_OUTPUT
	// Reset has been executed
	ResetDone:	BOOL; 
	// the axis is in target position
	MoveDone:	BOOL;
	// the axis hass jogged
	JogDone:	BOOL;
	// the axis has stopped
	StopDone: 	BOOL;
	// the axis was calibrated and has come to a standstill
	HomeDone:	BOOL;
	// the axis is ready
	Ready:		BOOL;
	// the command has been aborted
	CommandAborted: BOOL;
	// axis busy
	Busy: 		BOOL;
	// axis is moving
	Active: 	BOOL;
	// axis is stopping
	Stopping:	BOOL;
	// axis is standing still (no commands issued) this should be the default
	StandStill:	BOOL;
	// axis is in motion
	InMotion:	BOOL;
	// axis is homing
	Homing:		BOOL;
	// axis is Accelerating or Decelerating
	InRamp:		BOOL;
	// axis is tracking on position
	isTracking:	BOOL;
	//	error condition
	Error: 		BOOL;
	// number of error
	ErrorID: 	UDINT;
	// actual position of the axis
	ActualPosition: LREAL;
	// axis is calibrated;
	Calibrated:	BOOL := FALSE;
	
END_VAR
VAR
	Axis_Power:		MC_Power;
	Axis_Reset:		MC_Reset;
	Axis_Move:		MC_MoveAbsolute;
	Axis_Modulo:	MC_MoveModulo;
	//Axis_Position:	MC_ReadActualPosition;
	Axis_Stop:		MC_Stop;
	Axis_Status:	MC_ReadStatus;
	Axis_Home:		MC_Home;
	Axis_Jog: 		MC_Jog;
	Axis_SetpointEnable:	MC_ExtSetPointGenEnable;
	Axis_SetpointDisable:	MC_ExtSetPointGenDisable;
	StopAllowed:	BOOL;
	// Direction for Axis_SetpointFeed
	Direction:			DINT;
	// difference between set position and measured position
	PositionDifference:	LREAL;
	TrackPosition:		LREAL;
	TrackVelocity:		LREAL;
	TrackAcceleration:	LREAL;
END_VAR

VAR_IN_OUT
	// axis reference
	AxisRef:	AXIS_REF;
END_VAR

// query the status of the axis at the beginning of the cycle
Axis_Status(Enable := TRUE,
			Axis := AxisRef);

// Enable the axis (power signal or manual enable)
Axis_Power(
	Axis := AxisRef,
	Enable := Enable,
	Enable_Positive := Enable_Positive,
	Enable_Negative := Enable_Negative,
	Override := 100.0,
	Status => Ready);

Axis_Reset(
	Axis := 	AxisRef,
	Execute := 	Reset,
	Done => 	ResetDone);

(* Tracking section ********************************************** *)

IF Tracking THEN
	PositionDifference := LIMIT(-0.02, Position - ActualPosition, 0.02);
	TrackPosition := ActualPosition + PositionDifference;
	TrackVelocity := 0.0; // LIMIT(-1.0, 2.0 * Velocity, 1.0);
	TrackAcceleration := 0.0;
ELSE
	TrackPosition := ActualPosition;
	TrackVelocity := 0.0;
	TrackAcceleration := 0.0;
END_IF


IF NOT Tracking OR ABS(PositionDifference) < 1E-5 THEN // TrackVelocity = 0 AND TrackAcceleration = 0 THEN
	Direction := 0;
ELSIF PositionDifference < 0.0 THEN
	Direction := -1;
ELSE
	Direction := 1;
END_IF

isTracking := Tracking AND ABS(Position - ActualPosition) < 5.0E-3;
IF Tracking AND Ready AND Calibrated AND NOT StopAxis THEN
	Axis_SetpointEnable.Execute := TRUE;
ELSIF NOT Axis_SetpointEnable.Busy AND Axis_SetpointEnable.Done THEN
	Axis_SetpointEnable.Execute := FALSE;
END_IF

Axis_SetpointEnable(Axis := AxisRef,
	Position :=		TrackPosition,	// final destination
	PositionType := POSITIONTYPE_ABSOLUTE);
	
MC_ExtSetPointGenFeed(
	Position :=		TrackPosition,
	Velocity :=		TrackVelocity,
	Acceleration :=	TrackAcceleration,
	Direction :=	Direction, 
	Axis :=			AxisRef);

Axis_SetpointDisable(Axis := AxisRef,
	Execute := NOT Tracking);
	
(* end of tracking section  ********************************************** *)
	
IF isModuloAxis THEN
	Axis_Modulo( 
		Axis := 		AxisRef,
		Execute := 		MoveAxis AND Ready AND Calibrated,
		Position := 	Position,
		Velocity :=		Velocity,
		Direction := 	MC_Shortest_Way,
		Done => 		MoveDone);
ELSE
	Axis_Move( 
		Axis := 		AxisRef,
		Execute := 		MoveAxis AND Ready AND Calibrated,
		Position := 	Position,
		Velocity := 	Velocity,
		Done => 		MoveDone);
END_IF

Axis_Jog(
	JogForward := 	Jog_Forward AND Ready AND Enable_Positive,
	JogBackwards := Jog_Backwards AND Ready AND Enable_Negative,
	Mode := 		MC_JOGMODE_STANDARD_FAST,
	Done => 		JogDone, 
	Axis := 		AxisRef);

Axis_Home(
	Axis := 			AxisRef,
	Execute := 			HomeAxis AND Ready,
	Position := 		position, //DEFAULT_HOME_POSITION,
	HomingMode :=		HomingMode,
	bCalibrationCam := 	bCalibrationCam,
	Done => 			HomeDone);	
(*	
IF (MoveDone OR HomeDone OR JogDone) AND NOT Axis_Status.StandStill THEN
	StopAxis := TRUE;
END_IF
*)
IF MoveDone AND (NOT Axis_Modulo.Busy OR NOT Axis_Move.Busy) THEN
	MoveAxis := FALSE;
END_IF

IF JogDone THEN
	Jog_Forward := FALSE;
	Jog_Backwards := FALSE;
END_IF

IF HomeDone THEN
	Calibrated := TRUE;
	HomeAxis := FALSE;
END_IF

IF StopDone THEN
	StopAxis := FALSE;
END_IF

StopAllowed :=	Axis_Status.StandStill OR  
				Axis_Status.ContinuousMotion OR
				Axis_Status.DiscreteMotion OR
				Axis_Status.SynchronizedMotion OR
				Axis_Status.Homing;

Axis_Stop( 
	Axis := 	AxisRef,
	Execute := 	StopAxis AND StopAllowed,
	Done => 	StopDone);
(*
Axis_Position(
	Axis := 	AxisRef,
	Enable := 	Calibrated,
	Position => AbsolutePosition);
*)
IF isModuloAxis THEN
	ActualPosition := AxisRef.NcToPlc.ModuloActPos; // required e.g. for Filterwheel
ELSE
	ActualPosition := AxisRef.NcToPlc.ActPos;
END_IF

IF Axis_Power.Error THEN
	ErrorID := Axis_Power.ErrorID;
END_IF

IF Axis_SetpointEnable.Error THEN
	ErrorID := Axis_SetpointEnable.ErrorID;
END_IF

IF Axis_Reset.Error THEN
	ErrorID := Axis_Reset.ErrorID;
END_IF

IF Axis_Modulo.Error THEN
	ErrorID := Axis_Modulo.ErrorID;
END_IF

IF Axis_Move.Error THEN
	ErrorID := Axis_Move.ErrorID;
END_IF

IF Axis_Home.Error THEN
	ErrorID := Axis_Home.ErrorID;
END_IF

IF Axis_Jog.Error THEN
	ErrorID := Axis_Jog.ErrorID;
END_IF

IF Axis_Stop.Error THEN
	ErrorID := Axis_Stop.ErrorID;
END_IF

Busy := 	Axis_SetpointEnable.Busy OR
			Axis_Reset.Busy OR 
			Axis_Modulo.Busy OR
			Axis_Move.Busy OR 
			Axis_Home.Busy OR
			Axis_Jog.Busy;

Error := 	Axis_Power.Error OR 
			Axis_SetpointEnable.Error OR
			Axis_Reset.Error OR 
			Axis_Modulo.Error OR
			Axis_Move.Error OR 
			Axis_Home.Error OR
			Axis_Jog.Error OR 
			Axis_Stop.Error;

Active := 	// Axis_Power.Active OR //alsways true if enabled 
			Axis_Modulo.Active OR
			Axis_Move.Active OR 
			Axis_Home.Active OR
			Axis_Jog.Active OR 
			Axis_Stop.Active;

CommandAborted :=	Axis_Modulo.CommandAborted OR
					Axis_Move.CommandAborted OR 
					Axis_Home.CommandAborted OR
					Axis_Jog.CommandAborted OR 
					Axis_Stop.CommandAborted;	
	
IF NOT Error THEN
	ErrorID := 0;
END_IF
			
InMotion := Axis_Status.ConstantVelocity OR
			Axis_Status.DiscreteMotion OR
			Axis_Status.ContinuousMotion OR
			Axis_Status.SynchronizedMotion; 
InRamp :=	Axis_Status.Accelerating OR
			Axis_Status.Decelerating;
Stopping := Axis_Status.Stopping;
StandStill := Axis_Status.StandStill;
Homing :=	Axis_Status.Homing;
// InPosition := AxisRef.NcToPlc.TargetPos;

END_FUNCTION_BLOCK

// ---- POUs/HydraulicsControl.TcPOU
PROGRAM HydraulicsControl
VAR_INPUT
	// start the hydraulics
	enable:		BOOL := FALSE;
	// reset any hydraulics error
	reset: 		BOOL;
	// manual override to start the suction pump
	suction_manual:	BOOL;
	//manual override to stop the pump
	pump_manual_stop: BOOL;
END_VAR
VAR_OUTPUT
	// status of the brake: is the brake open?
	brake_open:			BOOL;
	// is the brake closed?
	brake_closed:		BOOL;
	// pump is running, but the pressure remains low
	pressure_failure:	BOOL;
	// suction was started, but it is not running
	suction_failure:	BOOL;
	// main pump is running but suction has a timeout
	hydraulics_failure:	BOOL;
	main_pump_failure: BOOL;
	// oil is low
	oil_low:			BOOL;
	// oil is high (unused?)
	oil_high:			BOOL;
	// oil pressure is 25 bars
	oil_pressure_OK:	BOOL;
	// oil is on reserve
	oil_warning:		BOOL;
	// oil filter is dirty
	oil_filter_dirty:	BOOL;
	// oil is below 10°C
	oil_cold:			BOOL;
	// oil is above 50°C
	oil_hot:			BOOL;
	// main pump is running
	pump_running:		BOOL;
	// suction pump is running
	suction_running :	BOOL := FALSE;
	// error condition
	error: 				BOOL;
END_VAR
VAR
	// command to open the brake
	iopen_brake:	BOOL := FALSE;
	// command to open the brake
	iclose_brake: BOOL;
	// monitors the pressure of the pump is running
	pressure_watchdog:	TON;
	// monitors the activation of the suction pump
	suction_watchdog: TON;
	// monitors the activation of the main pump
	main_pump_watchdog:	TON;
	// watch the hydraulics and suction pumps
	hydraulics_watchdog: TON;
	// represents the state of the main pump
	oil_pump_state:		RS;
	// represents the state of the brake
	brake_state: 		RS;
	// wait for the brake to open after pressure has been established
	brake_open_delay:	TON;
	// report brake opend after a short delay
	brake_opened_delay:	TON;
	// error state (set dominant)
	error_state:	SR;
	// trigger for suction pump
	suction_trigger:	SR;
	// timer to shut off hydraulics after break was closed
	hydraulics_off_timer:	TON  := (PT := T#300S);
	pan_maxiumum_trigger:	TON	:= (PT := T#10S);
	off_trigger:	F_TRIG;
	oil_level, last_oil_level:		REAL;
	oil_level_min:		REAL := 1.8;
	oil_level_max:		REAL := 2.8;
	HydraulicsLog,
	PumpLog,
	ReserveLog,
	oil_low_log,
	FilterLog,
	oil_max_log,
	OverTemperatureLog,
	UnderTemperatureLog,
	SuctionLog,
	HydraulicsFailureLog,
	BrakeClearingWarning,
	BrakeHydraulicsWarning,
	BrakeWarning: FB_EventLog;
	
	StatusWord, LastStatus:	UDINT;
END_VAR

(* 
Main control Logic for the Hydraulics system
* power on delay for main pump and suction pump
* start main pump if main control is ready (button pressed or remote)
* start suction pump if maximum in pan is reached
* suction pump runs for 60 seconds
* stop main pump if oil is low
* stop main pump if pressure fails for 10 seconds
*)
oil_low := NOT GVL_Hydraulics.oil_low;
oil_high := NOT GVL_Hydraulics.oil_high;
oil_warning := GVL_Hydraulics.oil_reserve;
oil_pressure_OK := GVL_Hydraulics.oil_pressure_OK;
oil_filter_dirty := NOT GVL_Hydraulics.oilfilter_dirty;
oil_cold := NOT GVL_Hydraulics.oil_undertemperature;
oil_hot := GVL_Hydraulics.oil_overtemperature;
oil_level := F_YREAL(GVL_Hydraulics.oil_level, 0, 16383, 0.0, 5.0);
pump_running := GVL_Hydraulics.pump_running;
suction_running := GVL_Hydraulics.suction_running;

pan_maxiumum_trigger(IN := GVL_Hydraulics.oilpan_maximum);

error_state(SET1 := pressure_failure OR	suction_failure OR hydraulics_failure OR oil_low OR main_pump_failure,
			RESET := reset,
			Q1 => error);
// clear reset, if no error present

IF NOT error THEN
	reset := FALSE;
END_IF

oil_pump_state(SET := enable,
				RESET1 := NOT enable OR error OR pump_manual_stop);

GVL_Hydraulics.oil_pump_enable := oil_pump_state.Q1;

(* This section controls the hydraulic brake responsible for azimuth and elevation. 
Especially the elevation is imbalanced if not in the position control loop. 
The brake must only be opened, if the elevation drive is activated concurrently.
*)


// close the brake if the pump is not running	
IF iclose_brake OR NOT pump_running THEN 
	iopen_brake := FALSE;
END_IF

// wait for pressure to build up (hack for oil_pressure_ok)
brake_open_delay(IN := pump_running AND oil_pressure_OK,
				PT := T#3S);
		
brake_state(SET := brake_open_delay.Q AND iopen_brake AND MAIN.brake_clearing,
			RESET1 := GVL_Telescope.azimut_limit_switch 
					  OR iclose_brake 
					  OR NOT pump_running
					  OR NOT MAIN.brake_clearing,
			Q1 => GVL_Telescope.brake_azimuth_eve);

// signal that the brake is open after one second
brake_opened_delay(	IN :=brake_state.Q1, 
					PT := T#1000MS,
					Q => brake_open);

brake_closed := NOT brake_open;
IF brake_closed THEN
	iclose_brake := FALSE;
END_IF
// turn off the hydraulics if the brake is closed and the pump is still running
hydraulics_off_timer(IN := brake_closed AND enable );
off_trigger(CLK := hydraulics_off_timer.Q);

IF hydraulics_off_timer.Q THEN
	enable := FALSE;
END_IF

(* This is the end of the brake control section *)

// adjust maximum oil level
IF (oil_level < oil_level_max AND GVL_Hydraulics.oilpan_maximum) OR 
	(oil_level > oil_level_max AND NOT GVL_Hydraulics.oilpan_maximum) THEN
	oil_level_max := oil_level;	
END_IF
suction_trigger(SET1 := GVL_Hydraulics.oilpan_maximum OR oil_level > oil_level_max,
				RESET := oil_level < oil_level_min);
GVL_Hydraulics.oil_suction_enable := suction_trigger.Q1 OR suction_manual;					
suction_watchdog(IN := GVL_Hydraulics.oil_suction_enable AND NOT suction_running,
					PT := T#15S,
					Q => suction_failure);
					
pressure_watchdog(IN := GVL_Hydraulics.oil_pump_enable AND 
						NOT oil_pressure_OK,
					PT := T#30S,
				  Q => pressure_failure);
hydraulics_watchdog(IN := pump_running AND NOT suction_running,
						PT := T#140S,
						Q => hydraulics_failure);

main_pump_watchdog(IN := GVL_Hydraulics.oil_pump_enable AND NOT pump_running,
					PT := T#10S,
					Q => main_pump_failure);

StatusWord.0 := oil_low;
StatusWord.1 := oil_high;
StatusWord.2 := oil_warning;
StatusWord.3 := oil_pressure_OK;
StatusWord.4 := oil_filter_dirty;
StatusWord.5 := oil_cold;
StatusWord.6 := oil_hot;
StatusWord.7 := brake_open;
StatusWord.8 := GVL_Main.brake_clearing;
StatusWord.9 := pump_running;
StatusWord.10 := suction_running;
StatusWord.11 := GVL_Hydraulics.oilpan_maximum;
StatusWord.12 := GVL_Hydraulics.oil_pump_enable;
StatusWord.13 := GVL_Hydraulics.oil_suction_enable;
IF ABS(last_oil_level - oil_level) > 0.02 THEN
	StatusWord.15 := TRUE;
	last_oil_level := oil_level;
ELSE
	StatusWord.15 := FALSE;
END_IF

IF StatusWord<>LastStatus THEN // publish new payload every second
	LastStatus := StatusWord;
	MAIN.MQTTClient.Publish('hydraulics', 'base', 'OilLow',			BOOL_TO_STRING(oil_low));
	MAIN.MQTTClient.Publish('hydraulics', 'base', 'OilHigh',		BOOL_TO_STRING(oil_high));
	MAIN.MQTTClient.Publish('hydraulics', 'base', 'OilMaximum',		BOOL_TO_STRING(GVL_Hydraulics.oilpan_maximum));
	MAIN.MQTTClient.Publish('hydraulics', 'base', 'OilReserve',		BOOL_TO_STRING(oil_warning));
	MAIN.MQTTClient.Publish('hydraulics', 'base', 'OilPressureOK', 	BOOL_TO_STRING(oil_pressure_OK));
	MAIN.MQTTClient.Publish('hydraulics', 'base', 'OilFilterDirty',	BOOL_TO_STRING(oil_filter_dirty));
	MAIN.MQTTClient.Publish('hydraulics', 'base', 'OilCold',		BOOL_TO_STRING(oil_cold));
	MAIN.MQTTClient.Publish('hydraulics', 'base', 'OilHot',			BOOL_TO_STRING(oil_Hot));
	MAIN.MQTTClient.Publish('hydraulics', 'base', 'BrakeOpen',		BOOL_TO_STRING(brake_open));
	MAIN.MQTTClient.Publish('hydraulics', 'base', 'BrakeClearing',	BOOL_TO_STRING(GVL_Main.brake_clearing));
	MAIN.MQTTClient.Publish('hydraulics', 'base', 'PumpRunning',	BOOL_TO_STRING(pump_running));
	MAIN.MQTTClient.Publish('hydraulics', 'base', 'SuctionRunning',	BOOL_TO_STRING(suction_running));
	MAIN.MQTTClient.Publish('hydraulics', 'base', 'OilLevel',		REAL_TO_STRING(oil_level));
	MAIN.MQTTClient.Publish('hydraulics', 'base', 'StatusWord',		UDINT_TO_STRING(StatusWord));
END_IF


				  				  
HydraulicsLog(Trigger := pressure_failure OR main_pump_failure,
				Level := ADSLOG_MSGTYPE_ERROR,
				FormatString := 'Main hydraulics pump / pressure: %s',
				OnMessage := 'FAILURE',
				OffMessage := 'OK',
				OffLevel := ADSLOG_MSGTYPE_HINT);

PumpLog(Trigger := pump_running,
				Level := ADSLOG_MSGTYPE_HINT,
				FormatString := 'Main hydraulics pump: %s',
				OnMessage := 'START',
				OffMessage := 'STOP',
				OffLevel := ADSLOG_MSGTYPE_HINT);
	
ReserveLog(Trigger := oil_warning,
			Level := ADSLOG_MSGTYPE_WARN,
			FormatString := 'oil reserve: %s',
			OnMessage := 'LOW',
			OffMessage := 'OK',
			OffLevel := ADSLOG_MSGTYPE_HINT);

oil_low_log(Trigger := oil_low,
				Level := ADSLOG_MSGTYPE_ERROR,
				FormatString := 'oil level: %s',
				OnMessage := 'LOW',
				OffMessage := 'OK',
				OffLevel := ADSLOG_MSGTYPE_HINT);

oil_max_log(Trigger := GVL_Hydraulics.oilpan_maximum,
				Level := ADSLOG_MSGTYPE_WARN,
				FormatString := 'oil level: %s',
				OnMessage := 'MAXIMUM',
				OffMessage := 'OK',
				OffLevel := ADSLOG_MSGTYPE_HINT);	
				
FilterLog(Trigger := oil_filter_dirty,
				Level := ADSLOG_MSGTYPE_WARN,
				FormatString := 'Hydraulics Filter is %s',
				OnMessage := 'dirty.');

OverTemperatureLog(Trigger := oil_hot,
				Level := ADSLOG_MSGTYPE_WARN,
				FormatString := 'Hydraulics Temperature is %s',
				OnMessage := 'high.');
				
UnderTemperatureLog(Trigger := oil_cold,
				Level := ADSLOG_MSGTYPE_WARN,
				FormatString := 'Hydraulics Temperature is %s',
				OnMessage := 'low.');

SuctionLog(Trigger := suction_failure,
				Level := ADSLOG_MSGTYPE_ERROR,
				FormatString := 'suction pump: %s',
				OnMessage := 'FAILURE',
				OffMessage := 'OK',
				OffLevel := ADSLOG_MSGTYPE_HINT);

HydraulicsFailureLog(Trigger := hydraulics_failure,
				Level := ADSLOG_MSGTYPE_ERROR,
				FormatString := 'suction pump while running main pump: %s',
				OnMessage := 'FAILURE',
				OffMessage := 'OK',
				OffLevel := ADSLOG_MSGTYPE_HINT);
				
BrakeClearingWarning(Trigger := NOT Main.brake_clearing AND iopen_brake,
				Level := ADSLOG_MSGTYPE_WARN,
				FormatString := '%s',
				OnMessage := 'Cannot open brake without brake clearing.');

BrakeWarning(	Trigger := brake_open,
				Level := ADSLOG_MSGTYPE_WARN,
				FormatString := '%s',
				OnMessage := 'Brake is open.',
				OffMessage := 'Brake is closed.');

BrakeHydraulicsWarning(Trigger := NOT enable AND iopen_brake,
				Level := ADSLOG_MSGTYPE_WARN,
				FormatString := '%s',
				OnMessage := 'Cannot open brake without running hydraulics.');

METHOD close_brake : BOOL
VAR_INPUT
END_VAR
// close the brake
iclose_brake := TRUE;

RETURN(brake_closed);
END_METHOD

METHOD open_brake : BOOL
VAR_INPUT
END_VAR
// start the pump
enable := TRUE;
// open the brake
IF oil_pressure_OK THEN
	iopen_brake := TRUE;
END_IF;
RETURN(brake_open);
END_METHOD

END_PROGRAM

// ---- POUs/MAIN.TcPOU
PROGRAM MAIN
VAR
	// telescope drives are ready to enable
	ready:				BOOL;
	// error stat on drive, power or hydraulics
	error:				BOOL;
	// manual, panel or remote reset
	reset:				BOOL;
	// start hydraulics
	start:				BOOL;
	// stop hydraulics 
	stop:				BOOL;
	// soft start trafo
	key_switch:			BOOL;
	//	open brake
	brake_clearing:		BOOL := FALSE;
	
	remote_start:		BOOL;
	remote_stop: 		BOOL;
	remote_reset:		BOOL;
	remote_keyswitch:	BOOL;
	remote_brake_clearing:	BOOL;
	// blink error lamp on warning
	error_lamp: 		FB_BLINK;
	power_lamp:			FB_BLINK;
	sound_horn:			FB_Horn;
	// main cabinet temperature in degrees
	cabinet_temperature:	REAL;
	// measures time between soft start command and power available
	ups_output_voltage:		REAL;
	ups_output_current:		REAL;
	ups_output_power:		REAL;
	PhaseLog:				FB_EventLog;
	TemperatureEvent,
	TemperatureCriticalEvent:	FB_EventLog;
	MQTTTimer : 		TON := (PT:=T#5S);
	GetHostName:		FB_GetHostName;
	HostName: 			STRING(255);
//	LightSwitch:		FB_ButtonEnable;
//	Lightbutton: 		BOOL;
	bExecute:			BOOL := TRUE;
	cabinet_temperature_warning:	SR;
	cabinet_temperature_critical:	SR;
	MQTTClient:		FB_MQTTCommunication;
	ups: 				PS_Q4_DcUpsEC_Cyclic_2;
	xActivate:			BOOL := TRUE;
	arrInputPD	AT%I*:	ARRAY[0..30] OF WORD;
	//UPS_Error,
	UPS_Alarm,
	UPS_Warning,
	UPS_BatMode,
	UPS_ReplaceBattery: FB_EventLog;
END_VAR

(* 
Main control loop
* Execute sub modules
* power management
* control panel switches and status lamps

* start switch activates Hydraulics and Trafo
* 
*)
GetHostName(bExecute := bExecute, sHostName => HostName);
bExecute := FALSE;
start := GVL_Main.start_switch OR remote_start;
stop := (NOT GVL_Main.stop_switch) OR remote_stop;
key_switch := GVL_Main.key_switch_remote OR remote_keyswitch;
brake_clearing := GVL_Main.brake_clearing OR remote_brake_clearing;
reset := GVL_Main.reset_switch OR GVL_pendant_control.reset_switch OR remote_reset;		
brake_clearing := NOT GVL_Main.brake_clearing;
cabinet_temperature := INT_TO_REAL(GVL_Main.main_cabinet_temperature) / 10.0;
cabinet_temperature_warning(SET1 := cabinet_temperature > 50.0,
							RESET := cabinet_temperature < 40.0);
cabinet_temperature_critical(SET1 := cabinet_temperature > 60.0,
							RESET := cabinet_temperature < 50.0);
IF key_switch THEN
	Transformer.start();
ELSE
	Transformer.stop();
END_IF

IF reset THEN
	Transformer.reset();
END_IF

IF start THEN
	HydraulicsControl.enable := TRUE;
END_IF
IF stop THEN
	HydraulicsControl.enable := FALSE;
END_IF

// telescope is ready when power available
ready :=  GVL_main.trafo_bypassed;

// QUINT UPS control section
ups(
	xActivate:= xActivate, 
	arrInputPD:= arrInputPD, 
	xActive=> , 
	xError=> , 
	wDiagCode=> , 
	wAddDiagCode=> , 
	wOutputVoltage=> ups_output_voltage, 
	wOutputCurrent=> ups_output_current, 
	xBatModeActive=> , 
	udtDataStruct=> , 
	xAlarm=> , 
	xWarning=> , 
	xReplaceBattery=> , 
	udtDiag=> );
	
ups_output_voltage := ups_output_voltage / 1000.0;
ups_output_current := ups_output_current / 1000.0;
ups_output_power := ups_output_voltage * ups_output_current;

PowerMonitoring();		
TelescopeControl();	//
CoverControl();	//
PendantControl();	//
NasmythControl();	//
HydraulicsControl();	//
ElevationControl();	//
AzimuthElevationControl();	//
DerotatorControl();	//
FilterWheelControl();	//
FocusControl();
MQTTClient();
Transformer();

error := GVL_Telescope.azimut_limit_switch
			OR FilterWheelControl.Error
			OR Focuscontrol.Error
			OR NasmythControl.error
			OR CoverControl.Error
			OR HydraulicsControl.error;
// set control lights					
GVL_Main.lamp_on_manual := PendantControl.manual;

IF GVL_Safety.Error THEN
	error_lamp.blink := e_blink.short;
ELSIF ElevationControl.error OR AzimuthElevationControl.error OR DerotatorControl.Error THEN
	error_lamp.blink := e_blink.long;
ELSIF HydraulicsControl.oil_warning OR HydraulicsControl.oil_hot OR HydraulicsControl.pressure_failure THEN
	error_lamp.blink := e_blink.slow;
ELSIF Transformer.error THEN
	error_lamp.blink := e_blink.fast;
ELSIF error THEN
	error_lamp.blink := e_blink.on;
ELSE
	error_lamp.blink := e_blink.off; 
END_IF

IF Transformer.restart_inhibited THEN
	power_lamp.blink := e_blink.short;
ELSIF GVL_main.trafo_bypassed THEN 
	power_lamp.blink := e_blink.on;
ELSIF Transformer.phase_available THEN
	power_lamp.blink := e_blink.long;
ELSIF NOT Transformer.phase_available THEN
	power_lamp.blink := e_blink.off;
ELSIF  Transformer.error THEN
	power_lamp.blink := e_blink.fast;
ELSE 
	power_lamp.blink := e_blink.off; 
END_IF
error_lamp(Q => GVL_Main.lamp_error);
//GVL_Main.lamp_error := error_lamp.Q;
power_lamp(Q => GVL_Main.lamp_power);
//GVL_Main.lamp_power := power_lamp.Q;

IF GVL_Telescope.azimut_limit_switch THEN
	sound_horn.horn := E_horn.long;
ELSIF Hydraulicscontrol.suction_failure THEN
	sound_horn.horn := E_horn.long;
ELSIF TelescopeControl.poweronwarning.Q THEN
	sound_horn.horn := E_horn.short;
ELSIF Pendantcontrol.horn THEN
	sound_horn.horn := E_horn.beep;
ELSE
	sound_horn.horn := E_horn.off;
END_IF 

sound_horn(Q => GVL_Telescope.horn );

SafetyHandling();

MQTTTimer(IN:=TRUE);
IF MQTTTimer.Q THEN // publish new payload every second
	MQTTTimer(IN:=FALSE);
	MQTTClient.Publish('electronics', 'base', 'MainCabinetTemperature', LREAL_TO_FMTSTR(cabinet_temperature, 2, TRUE));
	MQTTClient.Publish('electronics', 'base', 'PowerOK', BOOL_TO_STRING(Transformer.power_ok));
	MQTTClient.Publish('electronics', 'base', 'PhaseOK', BOOL_TO_STRING(Transformer.phase_available));
	MQTTClient.Publish('electronics', 'base', 'MainReady', BOOL_TO_STRING(ready));
	MQTTClient.Publish('electronics', 'base', 'MasterError', BOOL_TO_STRING(error));
	MQTTClient.Publish('electronics', 'base', 'UPSOutputVoltage', LREAL_TO_FMTSTR(ups_output_voltage, 3, TRUE));
	MQTTClient.Publish('electronics', 'base', 'UPSOutputCurrent', LREAL_TO_FMTSTR(ups_output_current, 3, TRUE));
	MQTTClient.Publish('electronics', 'base', 'UPSOutputPower', LREAL_TO_FMTSTR(ups_output_power, 3, TRUE));
	MQTTClient.Publish('electronics', 'base', 'UpsError', BOOL_TO_STRING(ups.xError));
	MQTTClient.Publish('electronics', 'base', 'UpsAlarm', BOOL_TO_STRING(ups.xAlarm));
	MQTTClient.Publish('electronics', 'base', 'UpsWarning', BOOL_TO_STRING(ups.xWarning));
	MQTTClient.Publish('electronics', 'base', 'UpsBatteryMode', BOOL_TO_STRING(ups.xBatModeActive));
	MQTTClient.Publish('electronics', 'base', 'UPSReplaceBattery', BOOL_TO_STRING(ups.xReplaceBattery));
END_IF

PhaseLog(	
	Trigger := 		NOT Transformer.phase_available, 
	Level := 		ADSLOG_MSGTYPE_ERROR,
	FormatString :=	'%s',
	OnMessage := 	'electrical phases:	ERROR!',
	OffLevel := 	ADSLOG_MSGTYPE_HINT,
	OffMEssage := 	'electrical phases:	active');
	
TemperatureEvent(	
	Trigger := 		cabinet_temperature_warning.Q1, 
	Level := 		ADSLOG_MSGTYPE_WARN,
	FormatString :=	'Main cabinet temperature warning:	%s',
	OnMessage := 	LREAL_TO_FMTSTR( cabinet_temperature, 1, TRUE),);
TemperatureCriticalEvent(	
	Trigger := 		cabinet_temperature_critical.Q1, 
	Level := 		ADSLOG_MSGTYPE_ERROR,
	FormatString :=	'Main cabinet temperature is critical:	%s!',
	OnMessage := 	LREAL_TO_FMTSTR( cabinet_temperature, 1, TRUE),);
(*	
UPS_Error(	
	Trigger := 		ups.xError, 
	Level := 		ADSLOG_MSGTYPE_ERROR,
	OnMessage := 	'UPS has an error!');
*)
UPS_Alarm(	
	Trigger := 		ups.xAlarm, 
	Level := 		ADSLOG_MSGTYPE_ERROR,
	OnMessage := 	'UPS has an alarm!');

	
UPS_Warning(	
	Trigger := 		ups.xWarning, 
	Level := 		ADSLOG_MSGTYPE_WARN,
	OnMessage := 	'UPS has a warning!');

UPS_BatMode(	
	Trigger := 		ups.xBatModeActive, 
	Level := 		ADSLOG_MSGTYPE_WARN,
	OnMessage := 	'UPS is on battery!');

UPS_ReplaceBattery(	
	Trigger := 		ups.xReplaceBattery, 
	Level := 		ADSLOG_MSGTYPE_WARN,
	OnMessage := 	'Replace UPS battery!');
(* 	NeutralCurrentGuardWarning		AT%I*:	BOOL;
	NeutralCurrentGuarError			AT%I*:	BOOL;
	ActivePowerGuardWarning			AT%I*:	BOOL;
	ActivePowerGuardError			AT%I*:	BOOL;
	ApparentPowerGuardWarning		AT%I*:	BOOL;
	ApparentPowerGuardError			AT%I*:	BOOL;
	ActivePower						AT%I*:	REAL;
	ActiveEnergy					AT%I*:	LINT;
	NeutralLineCurrent				AT%I*:	REAL; *)

END_PROGRAM

// ---- POUs/FunctionBlocks/FB_BLINK.TcPOU
FUNCTION_BLOCK FB_BLINK
VAR_INPUT
	blink:		E_Blink;
	ON_TIME:	TIME := T#500MS;
	OFF_TIME:	TIME := T#500MS;
END_VAR
VAR_OUTPUT
	Q:		BOOL;
END_VAR
VAR
    IMPULS   :TOF;
    PAUSE    :TOF;
END_VAR

CASE blink OF
	e_blink.slow:
		ON_TIME := T#500MS;
		OFF_TIME := T#500MS;
	e_blink.fast:
		ON_TIME := T#250MS;
		OFF_TIME := T#250MS;
	e_blink.short:
		ON_TIME := T#100MS;
		OFF_TIME := T#900MS;
	e_blink.long:
		ON_TIME := T#900MS;
		OFF_TIME := T#100MS;
END_CASE

IMPULS(IN:= NOT PAUSE.Q AND NOT IMPULS.Q, PT:= ON_TIME);
PAUSE(IN:= NOT PAUSE.Q AND NOT IMPULS.Q, PT:= OFF_TIME);
IF blink = e_blink.off THEN
	Q := FALSE;
ELSIF blink = e_blink.on THEN
	Q := TRUE;
ELSE
	Q := IMPULS.Q;	
END_IF

END_FUNCTION_BLOCK

// ---- POUs/FunctionBlocks/FB_Horn.TcPOU
FUNCTION_BLOCK FB_Horn
VAR_INPUT
	horn:	E_Horn;
END_VAR
VAR_OUTPUT
		Q:		BOOL;
END_VAR
VAR
	ON_TIME:	TIME := T#500MS;
	IMPULS   :TOF;
    PAUSE    :TOF;

END_VAR

CASE horn OF
	e_horn.off:
		ON_TIME := T#0MS;
	e_horn.beep:
		ON_TIME := T#500MS;
	e_horn.short:
		ON_TIME := T#5000MS;
	e_horn.long:
		ON_TIME := T#10000MS;
END_CASE

IMPULS(IN:= NOT PAUSE.Q AND NOT IMPULS.Q, PT:= ON_TIME);
IF horn = e_horn.off THEN
	Q := FALSE;
ELSE
	Q := IMPULS.Q;	
END_IF

END_FUNCTION_BLOCK

// ---- POUs/FunctionBlocks/FB_MQTTCommunication.TcPOU
FUNCTION_BLOCK FB_MQTTCommunication
VAR_INPUT
END_VAR
VAR_OUTPUT
END_VAR
VAR
	GetHostName:		FB_GetHostName;
	HostName: 			STRING(255);
    bSetParameter:		BOOL := FALSE;
    bConnect:			BOOL := FALSE;
    (* received message *)
	bSubscribed: 		BOOL;
	sTopicSub: 			STRING(255) := 'STELLA1/Telescope/SET';
	{attribute 'TcEncoding':='UTF-8'}
	sTopicRcv: 			STRING(255);
	{attribute 'TcEncoding':='UTF-8'}
	fbMessageQueue:		FB_IotMqttMessageQueue;
    fbMessage:			FB_IotMqttMessage;
	fbMqttClient:		FB_IotMqttClient;
	sPayloadRcv: 		STRING;
	influxMessage:		FB_InfluxMessage;
	measurement, 
	parameter, 
	value:		STRING(255);
END_VAR

(*
MQTT Communication section

Source:
https://infosys.beckhoff.com/english.php?content=../content/1033/tf6701_tc3_iot_communication_mqtt/3518541195.html&id=

*)
IF HostName='' THEN
	GetHostName.bExecute := TRUE;
ELSE
	GetHostName.bExecute := FALSE;
	bSetParameter := TRUE;
END_IF

GetHostName(sHostName => HostName);

// set the parameters once
IF bSetParameter THEN
    bSetParameter               := FALSE;
    fbMqttClient.sHostName      := '192.168.1.74';
    fbMqttClient.nHostPort      := 1883;
    fbMqttClient.sClientId      := HostName; 
    fbMqttClient.sTopicPrefix   := ''; 
	fbMqttClient.nKeepAlive     := 60; 
    fbMqttClient.ipMessageQueue := fbMessageQueue;
	bConnect := TRUE;
END_IF

// connect to the client
IF NOT fbMqttClient.bConnected THEN
;
END_IF

fbMqttClient.Execute(bConnect);
	
IF fbMqttClient.bConnected THEN
    IF NOT bSubscribed THEN
        bSubscribed := fbMqttClient.Subscribe(sTopic:=sTopicSub, 
												eQoS:=TcIotMqttQos.AtMostOnceDelivery);
    END_IF
END_IF

// receive queued messages
IF fbMessageQueue.nQueuedMessages > 0 THEN
    IF fbMessageQueue.Dequeue(fbMessage:=fbMessage) THEN
        fbMessage.GetTopic(pTopic:=ADR(sTopicRcv), nTopicSize:=SIZEOF(sTopicRcv) );
        fbMessage.GetPayload(pPayload:=ADR(sPayloadRcv), nPayloadSize:=SIZEOF(sPayloadRcv), bSetNullTermination:=TRUE);
		ADSLOGSTR( ADSLOG_MSGTYPE_HINT OR ADSLOG_MSGTYPE_LOG, 'MQTT %s', sPayloadRcv);
		IF sTopicRcv = sTopicSub THEN
			influxMessage(  sPayload := sPayloadRcv, measurement => measurement, parameter => parameter, value => value);
			IF NOT PendantControl.manual AND measurement = 'command' THEN
				IF parameter = 'power' THEN
					TelescopeControl.power := STRING_TO_BOOL(value);
				ELSIF parameter = 'park' THEN
					TelescopeControl.park := STRING_TO_BOOL(value);
				ELSIF parameter = 'gohome' THEN
					TelescopeControl.gohome := STRING_TO_BOOL(value);
				ELSIF parameter = 'track' THEN
					TelescopeControl.track := STRING_TO_BOOL(value);
				ELSIF parameter = 'goto' THEN
					TelescopeControl.goto := STRING_TO_BOOL(value);
				ELSIF parameter = 'slew' THEN
					TelescopeControl.slew := STRING_TO_BOOL(value);
				ELSIF parameter = 'stop' THEN
					TelescopeControl.stop := STRING_TO_BOOL(value);
				ELSIF parameter = 'reset' THEN
					TelescopeControl.reset := STRING_TO_BOOL(value);
				ELSIF parameter = 'masterreset' THEN
					ElevationControl.bSoEReset := STRING_TO_BOOL(value);
					AzimuthElevationControl.bSoEReset := STRING_TO_BOOL(value);
					DerotatorControl.bSoEReset := STRING_TO_BOOL(value);
				ELSIF parameter = 'nasmyth' THEN
					NasmythControl.left := STRING_TO_USINT(value) = 1;
					NasmythControl.right := STRING_TO_USINT(value) = 2;
				ELSIF parameter = 'rightascension' THEN
					TelescopeControl.track := FALSE;
					TelescopeControl.rightascension := STRING_TO_LREAL(value);
				ELSIF parameter = 'declination' THEN
					TelescopeControl.track := FALSE;
					TelescopeControl.declination := STRING_TO_LREAL(value);
				ELSIF parameter = 'elevation' THEN
					TelescopeControl.elevation := STRING_TO_LREAL(value);
				ELSIF parameter = 'azimuth' THEN
					TelescopeControl.azimuth := STRING_TO_LREAL(value);
				ELSIF parameter = 'focus' THEN
					FocusControl.position := STRING_TO_LREAL(value);
				ELSIF parameter = 'filter' THEN
					FilterWheelControl.filter_position := STRING_TO_USINT(value);
				ELSIF parameter = 'derotator' THEN
					TelescopeControl.track := FALSE;
					TelescopeControl.derotator_offset := STRING_TO_LREAL(value);
				ELSIF parameter = 'elevationoffset' THEN
					TelescopeControl.elevation_offset := STRING_TO_LREAL(value);
				ELSIF parameter = 'azimuthoffset' THEN
					TelescopeControl.azimuth_offset := STRING_TO_LREAL(value);
				ELSIF parameter = 'derotatoroffset' THEN
					TelescopeControl.derotator_offset := STRING_TO_LREAL(value);
				ELSIF parameter = 'resetpointing' THEN
					TelescopeControl.resetpointing  := STRING_TO_BOOL(value);
				ELSE
					ADSLOGSTR( ADSLOG_MSGTYPE_WARN OR ADSLOG_MSGTYPE_LOG, 'MQTT not understood %s', sPayloadRcv);
				END_IF
			END_IF // measurement
		END_IF // Topic
		sPayloadRcv := '';
    END_IF // Dequeue
END_IF

PROPERTY Error : BOOL
GET
Error := fbMqttClient.bError;
END_GET
END_PROPERTY

METHOD Publish : BOOL
VAR_INPUT
	domain: 	STRING(255) := 'environment';
	location: 	STRING(255) := 'roof';
	parameter:	STRING(255);
	value:		STRING(255);
END_VAR
VAR
	sPayloadPub: STRING(255) := '';
	fbFormat:	FB_FormatString;
	bError:		BOOL;
	nErrID: UDINT;
	retain_message:		BOOL := FALSE;
END_VAR
//sPayloadPub := 'environment,location=roof,host=CX-4E6032 ';
fbFormat( sFormat := '%s,location=%s,host=%s %s=%s', 
			arg1 := F_STRING(domain), 
			arg2 := F_STRING(location), 
			arg3 := F_STRING(HostName),
			arg4 := F_STRING(parameter),
			arg5 := F_STRING(value),
 
			sOut => sPayloadPub,
			bError => bError, 
			nErrID => nErrID );
// retain message if value is boolean
retain_message := value = 'TRUE' OR value = 'FALSE';

Publish := fbMqttClient.Publish(	
				sTopic:= 'STELLA1/Telemetry', 
				pPayload:= ADR(sPayloadPub), 
				nPayloadSize:= LEN2(ADR(sPayloadPub)),
				eQoS:= TcIotMqttQos.AtMostOnceDelivery,
				bRetain:= retain_message, 
				bQueue:= FALSE );
END_METHOD

METHOD PublishLog : BOOL
VAR_INPUT
	level: 	STRING(255) := 'INFO';
	message:	STRING(255);
	
END_VAR
VAR
	sPayloadPub: STRING(255) := '';
	fbFormat:	FB_FormatString;
	bError:		BOOL;
	nErrID: UDINT;
END_VAR
VAR_OUTPUT
	published: BOOL;
END_VAR
//sPayloadPub := 'environment,location=roof,host=CX-4E6032 ';
fbFormat( sFormat := 'log,host=%s,level=%s message="%s"', 
			arg1 := F_STRING(HostName), 
			arg2 := F_STRING(level), 
			arg3 := F_STRING(message),
 
			sOut => sPayloadPub,
			bError => bError, 
			nErrID => nErrID );

published := fbMqttClient.Publish(	
				sTopic:= 'STELLA1/Log', 
				pPayload:= ADR(sPayloadPub), 
				nPayloadSize:= LEN2(ADR(sPayloadPub)),
				eQoS:= TcIotMqttQos.AtMostOnceDelivery,
				bRetain:= FALSE, 
				bQueue:= FALSE );
END_METHOD

END_FUNCTION_BLOCK

// ---- POUs/TelescopeControl.TcPOU
PROGRAM TelescopeControl
VAR_INPUT
(*
TCS interface section
see https://gitlab.aip.de/bmk10k/telescope_firmware/snippets/5
*)
	
	// boolean, true: Power on, false: power off
	power: 		BOOL;
	// boolean, true: go to home position, unset track/goto if active
	gohome: 	BOOL;
	// boolean, true: go into park position, ready to stow telescope, unset track/goto
	park: 		BOOL;
	// boolean, TRUE: MOVE telescope TO last ra/de AND start tracking. Set 'goto' TO FALSE, IF TRUE. FALSE: Stop tracking as soon as possible
	track: 		BOOL;
	// boolean, TRUE: MOVE telescope TO tau/de AND stop there. Set track TO FALSE, IF TRUE. FALSE: no effect.)
	goto:		BOOL;	
	// move the telescope to a given az-alt position
	slew:		BOOL;
	// boolean, TRUE: Stop motion OF telescope immediately, set goto AND track TO FALSE. FALSE: Allow motion OF telescope again via track/goto).
	stop:		BOOL;	
	// initiates reset on all axis
	reset:		BOOL;
	// automatic tracking after goto
	autotrack:	BOOL := TRUE;
	// apparent right ascension, degrees, double
	rightascension:		LREAL := (4.0 + 35.0/60.0 + 54.09/3600.0) *15.0;	
	// apparent declination, degrees, double
	declination: 		LREAL := 16.0 + 30.0/60.0 + 25.4/3600.0;
	// desired elevation of the telescope pointing 
	elevation:	LREAL := 45.0;
	// desired azimut of the telescope pointing 
	azimuth:	LREAL := 320.0;
	// absolute offset for elevation
	elevation_offset:	LREAL := 0.0;
	// absolute offset for azimuth
	azimuth_offset : 	LREAL := 0.0;
	// absolute offset for time
	time_offset: 		LREAL := 0.0;
	// offset for the de-rotator
	derotator_offset:	LREAL := 0.0;
	// Nasmyth port 1 or 2
	Nasmyth_port: 		USINT;
	// reset pointing model
	resetpointing:		BOOL;
END_VAR
VAR
	// actual command from the TCS
	TCS_command: 	E_TCSCommand;
	// current Julian Date calculated from system time
	jd:				LREAL;
	// image derotation
	derotation_calc:	LREAL;
	// local siderial time calculated from Julian date
	lst:			LREAL;
	// elevation calulated when ra and dec are set by TCS
	elevation_calc:	LREAL; 
	// azimuth calulated when ra and dec are set by TCS
	azimuth_calc:	LREAL;
	// right ascension calulated when azimuth and elevation are set by TCS
	rightascension_calc:	LREAL;
	// declination calulated when azimuth and elevation are set by TCS
	declination_calc:		LREAL;
	// hour angle
	Hourangle_calc: LREAL;
	// precise astronomical	time
	fbTime: FB_AstroClock;
	
	eq2hor2:	FB_EQ2HOR2;
	hor2eq:		FB_HOR2EQ;
	
	// triggers power-failure event
	powerfailure: 	BOOL;
	// triggers power warning
	poweronwarning:	TP;
	// power on timeout
	power_timeout:	TON;
	// command timeout
	command_timeout:	TON;
	// tracking delay
	tracking_delay:	TON;
	// telescope is parked
	isparked:		BOOL;
	TCSpowerEvent,
	TCSgohomeEvent,
	TCSparkEvent,
	TCSgotoEvent,
	TCStrackEvent,
	TCSstopEvent,
	AltitudeEvent,
	TCSreadyEvent,
	TCSCTOEvent: FB_Eventlog;
	MQTTTimer : TON := (PT:=T#5S);
	// rotational velocity of the derotator
	DerotatorVelocity: LREAL;
	// rotational velocity of the elevation
	ElevationVelocity: LREAL;
	// rotational velocity of the elevation
	AzimuthVelocity: LREAL;
	// sign of derotation
	derotatation_sign: LREAL := 1.0;
	StatusWord, LastStatus:	UDINT;
END_VAR
VAR_OUTPUT
	//		TRUE, IF telescope can be operated
	ready:		BOOL; 
	// indicates an error on one of the components
	error:		BOOL;	
	//error id of axis
	errorid:	UDINT;	
	//TRUE, IF telescope is in fast-MOVE phase (includes pole-swap)
	sliding:	BOOL;	
	//TRUE, IF telescope is on tracking position AND currently tracking.
	tracking:	BOOL;	
	//TRUE, IF telescope is AT rest.
	stopped:	BOOL;	
	// true position of the elevation
	elevation_current:	LREAL;
	// true position of the azimuth
	azimuth_current:	LREAL;
	// true position of the de-rotator
	derotator_current:	LREAL;
	//	(time in sec. to reach the goto/track position)
	slewtime:			LREAL; 
	// True: telescope is calibrated
	homed:				BOOL;
	// telescope does not accept further commands
	busy:				BOOL;
END_VAR
VAR CONSTANT
// STELLA1
	// telescope site longitude, source: Google 
	longitude: 		LREAL := -16.50926; //13.101867;
	// telescope site latitude, source: Google
	latitude: 		LREAL := 28.30120; //52.404940;
	// telescope site height above sea level: estimated
	altitude: 		LREAL := 2390.0;
	elevation_park: LREAL := 60.0;
	azimuth_park: 	LREAL := 359.999;
	derotator_park: LREAL := 229.85;

	elevation_home: LREAL := 55.0;
	azimuth_home: 	LREAL := 180.0;
END_VAR
VAR PERSISTENT
	// azimuth axis offset/misalignment north-south
	AN_E:	LREAL;
	// azimuth axis offset/misalignment east-west
	AE_E:	LREAL;
	// gravitational flexure correction at the horizon
	TF:		LREAL;
	// collimation error of the electromagnetic axis
	BNP:	LREAL;
	// azimuth axis offset/misalignment north-south
	AN_A:	LREAL;
	// azimuth axis offset/misalignment east-west,
	AE_A:	LREAL;
	// Non-perpendicularity between the mount azimuth and elevation axes
	NPAE:	LREAL;
END_VAR

TelescopeAuxiliary();

// get the system time
fbTime();
jd := DateTime2JD(fbTime.time_RTCEX2);
lst := CT2LST(longitude, jd);
// set reset state either by hardware (key pressed) or by software (set by e.g. tcs)
IF GVL_Main.reset_switch THEN
	reset := TRUE;
END_IF


IF ElevationControl.error THEN
	errorid := ElevationControl.ErrorID;
	ElevationControl.reset := reset;
ELSIF AzimuthElevationControl.error THEN
	errorid := AzimuthElevationControl.ErrorID;
	AzimuthElevationControl.Reset := reset;
ELSIF FilterWheelControl.Error THEN
	errorid := FilterWheelControl.ErrorID;
	FilterWheelControl.Reset := reset;
ELSIF Focuscontrol.Error THEN
	errorid := Focuscontrol.ErrorID;
	FocusControl.reset := reset;
ELSIF DerotatorControl.Error THEN
	errorid := DerotatorControl.ErrorID;
	DerotatorControl.reset := reset;
END_IF

error := ElevationControl.error OR 
		 AzimuthElevationControl.error OR
		 FilterWheelControl.Error OR
		 Focuscontrol.Error OR
		 DerotatorControl.Error;

slewtime := MAX(MAX(ElevationControl.slewtime, AzimuthElevationControl.slewtime), DerotatorControl.slewtime);
			
IF error THEN
	gohome := 	FALSE;
	track := 	FALSE;
	goto := 	FALSE;
	slew := 	FALSE;
ELSE
	errorid := 0;
END_IF

IF ElevationControl.error THEN
	ElevationControl.enable := FALSE;
	AzimuthElevationControl.enable := FALSE;
	HydraulicsControl.close_brake();
END_IF

eq2hor2(alpha := rightascension,
	delta := declination,
	lon := longitude,
	lat := latitude,
	JD := jd + time_offset,
	alt => elevation_calc,
	az => azimuth_calc,
	ha => hourangle_calc);

// apply pointing model
elevation_calc := elevation_calc + PointingModelElevation(azimuth_calc, elevation_calc, elevation_offset, AN_E, AE_E, TF);
azimuth_calc := azimuth_calc + PointingModelAzimuth(azimuth_calc, elevation_calc, azimuth_offset, BNP, AN_A, AE_A, NPAE);
// calculate derotator position 
derotation_calc := F_DerotatorPosition2(azimuth_calc, elevation_calc, declination_calc, latitude, derotatation_sign)  + derotator_offset;
// calculate velocities
DerotatorVelocity := F_Derotatorvelocity(elevation_calc, azimuth_calc, latitude);
ElevationVelocity := F_Elevationvelocity(azimuth_calc, latitude);
AzimuthVelocity := F_Azimuthvelocity(elevation_calc, azimuth_calc, latitude);

IF (azimuth_calc > 310.0 AND AzimuthVelocity > 0.0) OR (azimuth_calc > 440.0) THEN
	azimuth_calc := azimuth_calc - 360.0;
ELSIF (azimuth_calc < 80.0 AND AzimuthVelocity < 0.0) OR (azimuth_calc < -50.0) THEN
	azimuth_calc := azimuth_calc + 360.0;
END_IF

IF (derotation_calc > 290.0 AND DerotatorVelocity > 0.0) OR (derotation_calc > 380.0) THEN
	derotation_calc := derotation_calc - 360.0;
ELSIF (derotation_calc < 20.0 AND DerotatorVelocity < 0.0) OR (derotation_calc < -70.0) THEN
	derotation_calc := derotation_calc + 360.0;
END_IF
// get current coordinates	
azimuth_current := AzimuthElevationControl.act_position;
elevation_current := ElevationControl.actual_position;
derotator_current := DerotatorControl.actual_position;

IF resetpointing THEN
	AN_A := 0.0;
	AN_E := 0.0;
	AE_A := 0.0;
	AE_E := 0.0;
	BNP := 0.0;
	TF := 0.0;
	NPAE := 0.0;
	resetpointing := FALSE;
END_IF

// calculate equatorial coordinates
hor2eq(alt := elevation_current - PointingModelElevation(azimuth_calc, elevation_calc, elevation_offset, AN_E, AE_E, TF), 
		az := azimuth_current - PointingModelAzimuth(azimuth_calc, elevation_calc, azimuth_offset, BNP, AN_A, AE_A, NPAE),
		jd := jd,
		lat := latitude,
		lon := longitude,
		altitude := altitude,
		ra => rightascension_calc,
		dec => declination_calc);		
	
poweronwarning(IN := power, PT := T#10S);

power_timeout(IN := TCS_command = E_TCSCommand.no_command AND NOT isparked, PT := T#12H);
command_timeout();
IF power_timeout.Q AND NOT isparked THEN
	park := TRUE;
END_IF

IF Nasmyth_port = 1 THEN
	NasmythControl.right := FALSE;
	IF NasmythControl.Nasmyth_left THEN
		NasmythControl.left := FALSE;
		NasmythControl.enable := FALSE;
	ELSE
		NasmythControl.left := TRUE;
		NasmythControl.enable := TRUE;
	END_IF
ELSIF Nasmyth_port = 2 THEN
	NasmythControl.left := FALSE;
    IF NasMythControl.Nasmyth_right THEN
		NasmythControl.right := FALSE;
		NasmythControl.enable := FALSE;
	ELSE
		NasmythControl.right := TRUE;
		NasmythControl.enable := TRUE;
	END_IF
ELSE
	NasmythControl.right := FALSE;
	NasmythControl.left := FALSE;
	NasmythControl.enable := FALSE;	
END_IF
	
		
// set TCS_command according to state variables ordered by precedence
IF power THEN
	TCS_command := E_TCSCommand.poweron;
ELSIF stop THEN
	TCS_command := E_TCSCommand.stop;
	goto := FALSE;
	track := FALSE;
	slew := FALSE;
	gohome := FALSE;
	park := FALSE;
ELSIF park THEN
	goto := FALSE;
	track := FALSE;
	slew := FALSE;
	gohome := FALSE;
	IF ready AND stopped THEN
		TCS_command := E_TCSCommand.park;
	END_IF
ELSIF gohome THEN
	park := FALSE;
	goto := FALSE;
	track := FALSE;
	slew := FALSE;
	IF ready AND NOT busy AND stopped THEN
		TCS_command := E_TCSCommand.gohome;
	END_IF
ELSIF goto THEN
	track := FALSE;
	slew := FALSE;
	IF ready AND NOT busy THEN
		TCS_command := E_TCSCommand.goto;
	END_IF
ELSIF slew THEN
	goto := FALSE;
	track := FALSE;
	IF ready AND NOT busy THEN
		TCS_command := E_TCSCommand.slew;
	END_IF
ELSIF track THEN
	goto := FALSE;
	slew := FALSE;
	IF ready AND NOT busy THEN
		TCS_command := E_TCSCommand.track;
	END_IF
ELSE
	TCS_command := E_TCSCommand.no_command;
	ElevationControl.MoveAxis := FALSE;
	AzimuthElevationControl.MoveAxis := FALSE;
	DerotatorControl.MoveAxis := FALSE;
	ElevationControl.Tracking := FALSE;
	AzimuthElevationControl.Tracking := FALSE;
	DerotatorControl.Tracking := FALSE;
END_IF

IF TCS_command = E_TCSCommand.poweron THEN
	poweron();
	command_timeout(IN := TCS_command = E_TCSCommand.poweron, PT := T#12H);
	TCSCTOEvent.OnMessage := 'POWER';
ELSIF TCS_command = E_TCSCommand.stop THEN
	stoptelescope();
	command_timeout(IN := TCS_command = E_TCSCommand.stop, PT := T#2S);
	TCSCTOEvent.OnMessage := 'STOP';
ELSIF TCS_command = E_TCSCommand.park THEN
	parktelescope();
	command_timeout(IN := TCS_command = E_TCSCommand.park, PT := T#2M);
	TCSCTOEvent.OnMessage := 'PARK';
ELSIF TCS_command = E_TCSCommand.gohome THEN
	hometelescope();
	command_timeout(IN := TCS_command = E_TCSCommand.gohome, PT := T#2M);
	TCSCTOEvent.OnMessage := 'GOHOME';
ELSIF TCS_command = E_TCSCommand.goto THEN
	gototelescope();
	command_timeout(IN := TCS_command = E_TCSCommand.goto, PT := T#2M);
	TCSCTOEvent.OnMessage := 'GOTO';
ELSIF TCS_command = E_TCSCommand.slew THEN
	slewtelescope();
	command_timeout(IN := TCS_command = E_TCSCommand.slew, PT := T#2M);
	TCSCTOEvent.OnMessage := 'SLEW';
ELSIF TCS_command = E_TCSCommand.track THEN
	tracktelescope();
	command_timeout(IN := TCS_command = E_TCSCommand.track, PT := T#12H);
	TCSCTOEvent.OnMessage := 'TRACK';
ELSE
	// disable command timeout
	command_timeout(IN := FALSE);
	TCSCTOEvent.OnMessage := 'NOCOMMAND';
END_IF
 
sliding := NOT tracking AND (ElevationControl.ElevationAxis.InMotion OR ElevationControl.ElevationAxis.InRamp OR
			AzimuthElevationControl.AzimuthAxis.InMotion OR AzimuthElevationControl.AzimuthAxis.InRamp OR
			DerotatorControl.DerotatorAxis.InMotion OR DerotatorControl.DerotatorAxis.InRamp);

// signal must be stable for 5500MS			
tracking_delay(in := ElevationControl.ElevationAxis.isTracking AND 
			AzimuthElevationControl.AzimuthAxis.isTracking AND
			DerotatorControl.DerotatorAxis.isTracking,PT :=T#5500MS, Q => tracking);
			
stopped :=  (NOT ElevationControl.enable OR ElevationControl.ElevationAxis.StandStill) AND 
			(NOT AzimuthElevationControl.Enable OR AzimuthElevationControl.AzimuthAxis.StandStill) AND
			(NOT DerotatorControl.enable OR DerotatorControl.DerotatorAxis.StandStill);
			
homed := ElevationControl.Calibrated AND
			AzimuthElevationControl.calibrated AND
			FilterWheelControl.Calibrated AND
			FocusControl.Calibrated AND
			DerotatorControl.Calibrated;
			
ready := homed AND 
	CoverControl.isopen AND 
	ElevationControl.enable AND
	AzimuthElevationControl.enable AND
	DerotatorControl.enable AND HydraulicsControl.brake_open AND 
    NOT error;

busy := ElevationControl.ElevationAxis.Busy OR
		AzimuthElevationControl.AzimuthAxis.Busy OR
		DerotatorControl.DerotatorAxis.Busy OR
		FocusControl.FocusAxis.Busy OR
		FilterWheelControl.FilterWheelAxis.Busy;
		
// unset the STOP command if telescope is already stopped
IF stopped THEN
	stop := FALSE;
END_IF
	
IF NOT error THEN
	reset := FALSE;
END_IF

IF SafetyHandling.Emergency_stop THEN
	ElevationControl.enable := FALSE;
	AzimuthElevationControl.enable := FALSE;
	DerotatorControl.enable := FALSE;
END_IF
IF sliding OR track OR tracking THEN
	MQTTTimer.PT := T#1000MS;
ELSE
	MQTTTimer.PT := T#5000MS;
END_IF
MQTTTimer(IN:=TRUE);
IF MQTTTimer.Q THEN // publish new payload every second
	MQTTTimer(IN:=FALSE);

	MAIN.MQTTClient.Publish('telescope', 'dome', 'JulianDate', LREAL_TO_STRING(jd));
	MAIN.MQTTClient.Publish('telescope', 'dome', 'LocalSiderialTime', LREAL_TO_STRING(lst));
	MAIN.MQTTClient.Publish('telescope', 'dome', 'Azimuth', LREAL_TO_STRING(azimuth_current));
	MAIN.MQTTClient.Publish('telescope', 'dome', 'Elevation', LREAL_TO_STRING(elevation_current));
	MAIN.MQTTClient.Publish('telescope', 'dome', 'Derotator', LREAL_TO_STRING(derotator_current));
	MAIN.MQTTClient.Publish('telescope', 'dome', 'HourAngle', LREAL_TO_STRING(hourangle_calc));
	MAIN.MQTTClient.Publish('telescope', 'dome', 'RightAscension', LREAL_TO_STRING(rightascension_calc));
	MAIN.MQTTClient.Publish('telescope', 'dome', 'Declination', LREAL_TO_STRING(declination_calc));
	MAIN.MQTTClient.Publish('telescope', 'dome', 'azimuth_offset', LREAL_TO_STRING(azimuth_offset));
	MAIN.MQTTClient.Publish('telescope', 'dome', 'elevation_offset', LREAL_TO_STRING(elevation_offset));
	MAIN.MQTTClient.Publish('telescope', 'dome', 'derotator_torque', LREAL_TO_STRING(DerotatorControl.derotator_torque));
	MAIN.MQTTClient.Publish('telescope', 'dome', 'elevation_torque', LREAL_TO_STRING(ElevationControl.elevation_torque));
	MAIN.MQTTClient.Publish('telescope', 'dome', 'azimuth_torque', LREAL_TO_STRING(AzimuthElevationControl.azimuth_torque));
	
	MAIN.MQTTClient.Publish('telescope', 'dome', 'errorid',		UDINT_TO_STRING(errorid));
	MAIN.MQTTClient.Publish('telescope', 'dome', 'error',		BOOL_TO_STRING(error));
	MAIN.MQTTClient.Publish('telescope', 'dome', 'ready',		BOOL_TO_STRING(ready));
	MAIN.MQTTClient.Publish('telescope', 'dome', 'busy',		BOOL_TO_STRING(busy));
	MAIN.MQTTClient.Publish('telescope', 'dome', 'sliding',		BOOL_TO_STRING(sliding));
	MAIN.MQTTClient.Publish('telescope', 'dome', 'tracking', 	BOOL_TO_STRING(tracking));
	MAIN.MQTTClient.Publish('telescope', 'dome', 'stopped',		BOOL_TO_STRING(stopped));
	MAIN.MQTTClient.Publish('telescope', 'dome', 'homed',		BOOL_TO_STRING(homed));
END_IF

StatusWord.0 := error;
StatusWord.1 := ready;
StatusWord.2 := sliding;
StatusWord.3 := tracking;
StatusWord.4 := stopped;
StatusWord.5 := homed;
StatusWord.6 := power;
StatusWord.7 := park;
StatusWord.8 := gohome;
StatusWord.9 := track;
StatusWord.10 := goto;
StatusWord.11 := slew;
StatusWord.12 := stop;
StatusWord.13 := busy;

IF StatusWord<>LastStatus THEN // publish new payload every second
	LastStatus := StatusWord;
	MAIN.MQTTClient.Publish('telescope', 'dome', 'error',		BOOL_TO_STRING(error));
	MAIN.MQTTClient.Publish('telescope', 'dome', 'ready',		BOOL_TO_STRING(ready));
	MAIN.MQTTClient.Publish('telescope', 'dome', 'sliding',		BOOL_TO_STRING(sliding));
	MAIN.MQTTClient.Publish('telescope', 'dome', 'tracking', 	BOOL_TO_STRING(tracking));
	MAIN.MQTTClient.Publish('telescope', 'dome', 'stopped',		BOOL_TO_STRING(stopped));
	MAIN.MQTTClient.Publish('telescope', 'dome', 'homed',		BOOL_TO_STRING(homed));
	MAIN.MQTTClient.Publish('telescope', 'dome', 'power',		BOOL_TO_STRING(power));
	MAIN.MQTTClient.Publish('telescope', 'dome', 'park',		BOOL_TO_STRING(park));
	MAIN.MQTTClient.Publish('telescope', 'dome', 'gohome',		BOOL_TO_STRING(gohome));
	MAIN.MQTTClient.Publish('telescope', 'dome', 'track',		BOOL_TO_STRING(track));
	MAIN.MQTTClient.Publish('telescope', 'dome', 'goto',		BOOL_TO_STRING(goto));
	MAIN.MQTTClient.Publish('telescope', 'dome', 'slew',		BOOL_TO_STRING(slew));
	MAIN.MQTTClient.Publish('telescope', 'dome', 'stop',		BOOL_TO_STRING(stop));
	MAIN.MQTTClient.Publish('telescope', 'dome', 'busy',		BOOL_TO_STRING(busy));
END_IF


(* Event function blocks start here. *)
TCSpowerEvent(	Trigger := powerfailure, 
				Level := ADSLOG_MSGTYPE_ERROR,
				FormatString := 'power %s',
				OnMessage := 'Failure',
				OffMessage := 'OK');

TCSgohomeEvent(	Trigger := gohome, 
				Level := ADSLOG_MSGTYPE_HINT,
				FormatString := 'GOHOME %s',
				OnMessage := 'commencing',
				OffMEssage := 'completed');
TCSparkEvent(	Trigger := park, 
				Level := ADSLOG_MSGTYPE_HINT,
				FormatString := 'PARK %s',
				OnMessage := 'commencing',
				OffMEssage := 'completed');
TCSgotoEvent(	Trigger := goto, 
				Level := ADSLOG_MSGTYPE_HINT,
				FormatString := 'GOTO %s',
				OnMessage := 'commencing',
				OffMEssage := 'completed');
TCStrackEvent(	Trigger := track, 
				Level := ADSLOG_MSGTYPE_HINT,
				FormatString := 'TRACK %s',
				OnMessage := 'commencing',
				OffMEssage := 'completed');
TCSstopEvent(	Trigger := stop, 
				Level := ADSLOG_MSGTYPE_WARN,
				FormatString := 'STOP %s',
				OnMessage := 'commencing',
				OffMEssage := 'completed',
				OffLevel := ADSLOG_MSGTYPE_HINT);
AltitudeEvent(	Trigger := power AND elevation_calc<0.0, 
				Level := ADSLOG_MSGTYPE_WARN,
				FormatString := '%s',
				OnMessage := 'Target below horizon',
				OffMEssage := '');
TCSreadyEvent(	Trigger := power AND ready, 
				Level := ADSLOG_MSGTYPE_HINT,
				FormatString := '%s',
				OnMessage := 'STELLA1 startup finished');
TCSCTOEvent(	Trigger := command_timeout.Q, 
				Level := ADSLOG_MSGTYPE_WARN,
				FormatString := 'A timeout occured during %s command!',
				OnMessage := 'NOCOMMAND');

METHOD gototelescope: USINT
VAR_INPUT
END_VAR
VAR
	GoToEvent:	FB_Eventlog;
	command_timeout:	TON;
END_VAR
VAR_STAT
	Stage:		USINT := 0;
	LastStage:	USINT := 101;
END_VAR
gototelescope := Stage;
command_timeout(IN := Stage < 100, PT := T#600S);
IF command_timeout.Q THEN
	error := TRUE;
	errorid := 16#10;
	goto := FALSE;
	Stage := 0;
	RETURN;
END_IF

IF elevation_calc<2.0 THEN
	error := TRUE;
	errorid := 16#15;
	goto := FALSE;
	Stage := 0;
	RETURN;
END_IF

IF reset OR error THEN
	Stage := 0;
	RETURN;
END_IF

CASE Stage OF
	0:	
		IF ready AND NOT busy THEN
			Stage := 25;
		END_IF
	25:	
		ElevationControl.position := elevation_calc;
		AzimuthElevationControl.position := azimuth_calc;
		DerotatorControl.position := derotation_calc;
		DerotatorControl.Velocity := 10.0;
		ElevationControl.velocity := 10.0;
		AzimuthElevationControl.velocity := 10.0;
		
		ElevationControl.MoveAxis := TRUE;
		AzimuthElevationControl.MoveAxis := TRUE;
		DerotatorControl.MoveAxis := TRUE;
		IF ElevationControl.ElevationAxis.Busy AND
			AzimuthElevationControl.AzimuthAxis.Busy AND
			DerotatorControl.DerotatorAxis.Busy THEN
				Stage := 50;
		END_IF
	50:
		IF NOT ElevationControl.ElevationAxis.Busy AND ElevationControl.ElevationAxis.MoveDone THEN
			ElevationControl.MoveAxis := FALSE;
		END_IF
		IF NOT AzimuthElevationControl.AzimuthAxis.Busy AND AzimuthElevationControl.AzimuthAxis.MoveDone THEN
			AzimuthElevationControl.MoveAxis := FALSE;
		END_IF
		IF NOT DerotatorControl.DerotatorAxis.Busy AND DerotatorControl.DerotatorAxis.MoveDone THEN
			DerotatorControl.MoveAxis := FALSE;
		END_IF
		IF NOT ElevationControl.MoveAxis AND 
           NOT AzimuthElevationControl.MoveAxis AND 
		   NOT DerotatorControl.MoveAxis THEN
		   Stage := 75;
		END_IF
	75:
		IF NOT sliding AND stopped THEN // all axis standstill
			Stage := 100;
		END_IF
	100:
		ElevationControl.MoveAxis := FALSE;
		AzimuthElevationControl.MoveAxis := FALSE;
		DerotatorControl.MoveAxis := FALSE;
		azimuth := azimuth_calc;
		elevation := elevation_calc;
		goto := FALSE;
		// enable automatic tracking
		track := autotrack;
		Stage := 0;
END_CASE
GoToEvent(Trigger := Stage > LastStage, FormatString := 'GoTo progress: %s', OnMessage := USINT_TO_STRING(Stage));
LastStage := Stage;
END_METHOD

METHOD hometelescope : BOOL
VAR_INPUT
END_VAR

VAR
	HomeEvent: FB_Eventlog;
	command_timeout: TON;
END_VAR
command_timeout(IN := NOT hometelescope, PT := T#600S);
IF command_timeout.Q THEN
	error := TRUE;
	errorid := 16#30;
	hometelescope :=TRUE;
END_IF

IF ready AND stopped AND NOT busy AND NOT tracking THEN
	ElevationControl.velocity := 10.0;
	ElevationControl.position := elevation_home;
	ElevationControl.MoveAxis := TRUE;
	AzimuthElevationControl.velocity := 10.0;
	AzimuthElevationControl.position := azimuth_home;
	AzimuthElevationControl.MoveAxis := TRUE;
	DerotatorControl.Velocity := 10.0;
	DerotatorControl.position := 180.0;
	DerotatorControl.MoveAxis := TRUE;	
END_IF

IF ElevationControl.ElevationAxis.MoveDone AND 
	AzimuthElevationControl.AzimuthAxis.MoveDone AND 
	DerotatorControl.DerotatorAxis.MoveDone THEN
	gohome := FALSE;
	elevation := elevation_current;
	azimuth := azimuth_current;
	hometelescope := TRUE;
ELSE
	hometelescope := FALSE;
END_IF

HomeEvent(Trigger := hometelescope, 
			Level := ADSLOG_MSGTYPE_HINT,
			FormatString := '%s',
			OnMessage := 'Telescope is homed.');
END_METHOD

METHOD parktelescope: USINT
VAR_INPUT
END_VAR
VAR
	ParkEvent:	FB_Eventlog;
END_VAR
VAR_STAT
	Stage:		USINT := 0;
	LastStage:	USINT := 101;
END_VAR
parktelescope := Stage;
IF reset OR error THEN
	Stage := 0;
END_IF
IF isparked THEN
	Stage := 100;
END_IF
CASE Stage OF
	0: 
		gohome := 	FALSE;
		track := 	FALSE;
		goto := 	FALSE;
		slew := 	FALSE;
		Focuscontrol.position := 53.6;
		FilterWheelControl.filter_position := 0;
		//FilterWheelControl.Enable := FALSE;
		IF Error THEN // emergency park
			HydraulicsControl.close_brake();
			ElevationControl.enable := FALSE;
			AzimuthElevationControl.Enable := FALSE;
			DerotatorControl.enable := FALSE;	
			CoverControl.close := TRUE;	
			Stage := 80;
		END_IF
		Stage := 20;
	20:
		ElevationControl.position := elevation_park;
		ElevationControl.velocity := 10.0;
		ElevationControl.MoveAxis := TRUE;
		AzimuthElevationControl.position := azimuth_park;
		AzimuthElevationControl.velocity := 10;
		AzimuthElevationControl.MoveAxis := TRUE;
		DerotatorControl.position := derotator_park;
		DerotatorControl.Velocity := 10.0;
		DerotatorControl.MoveAxis := TRUE;
		IF ElevationControl.ElevationAxis.Busy AND
			AzimuthElevationControl.AzimuthAxis.Busy AND
			DerotatorControl.DerotatorAxis.Busy THEN
				Stage := 40;
		END_IF
	40:
		IF ElevationControl.ElevationAxis.MoveDone THEN
			ElevationControl.MoveAxis := FALSE;
		END_IF
		IF AzimuthElevationControl.AzimuthAxis.MoveDone THEN
			AzimuthElevationControl.MoveAxis := FALSE;
		END_IF
		IF DerotatorControl.DerotatorAxis.MoveDone THEN
			DerotatorControl.MoveAxis := FALSE;
		END_IF
		IF NOT sliding THEN // all axis standstill
			Stage := 60;
		END_IF
	60:
		IF NOT ElevationControl.enable AND NOT AzimuthElevationControl.Enable AND NOT DerotatorControl.enable THEN
			stage := 80;
		END_IF
		
		IF stopped THEN 
			ElevationControl.enable := FALSE;
			AzimuthElevationControl.Enable := FALSE;
			DerotatorControl.enable := FALSE;
		END_IF
		
		ElevationControl.MoveAxis := FALSE;
		AzimuthElevationControl.MoveAxis := FALSE;
		DerotatorControl.MoveAxis := FALSE;
	80:
		IF ElevationControl.enable OR AzimuthElevationControl.Enable OR DerotatorControl.enable THEN
			stage := 60;
		END_IF
		IF HydraulicsControl.brake_closed THEN
			CoverControl.close := TRUE;
			HydraulicsControl.enable := FALSE;			
		END_IF
		IF CoverControl.isclosed THEN
			Stage := 100;
		END_IF
	100:
			isparked := TRUE;
			park := FALSE;
			parktelescope := 100;
			Stage := 0;	
END_CASE
ParkEvent(Trigger := Stage > LastStage, FormatString := 'Parking progress: %s', OnMessage := USINT_TO_STRING(Stage));
LastStage := Stage;
END_METHOD

METHOD poweron : BOOL
VAR_INPUT
END_VAR
VAR
END_VAR
IF NOT Main.brake_clearing THEN
	powerfailure := TRUE;
	TCSpowerEvent.OnMessage := 'failure: brake clearing not set';
	power := FALSE;
ELSIF NOT Transformer.power_OK THEN
	powerfailure := TRUE;
	TCSpowerEvent.OnMessage := 'failure: main power failure';
	power := FALSE;
ELSIF NOT Transformer.phase_available THEN
	powerfailure := TRUE;
	TCSpowerEvent.OnMessage := 'failure: hydraulics power failure';
	power := FALSE;
ELSIF error THEN
	powerfailure := TRUE;
	TCSpowerEvent.OnMessage := 'Generic error during power on occured.';
	power := FALSE;
ELSE
	powerfailure := FALSE;		
END_IF
// COVER MUST BE OPENED FOR A SUCCESSFUL WAKE & SHAKE COMMAND!
Covercontrol.open := TRUE;

